LIN {X 0,Y 431.61,Z 997.566,A -85,B 0,C 180,E1 -9443.457,E2 -9443.457} C_VEL
LIN {X 0,Y 431.611,Z 1001.678,A -85,B 0,C 180,E1 -9444.864,E2 -9444.864} C_VEL
LIN {X 0,Y 431.653,Z 1004.723,A -85,B 0,C 180,E1 -9446.268,E2 -9446.268} C_VEL
LIN {X 0,Y 431.594,Z 1006.161,A -85,B 0,C 180,E1 -9447.202,E2 -9447.202} C_VEL
LIN {X 0,Y 431.598,Z 1007.192,A -85,B 0,C 180,E1 -9448.135,E2 -9448.135} C_VEL
LIN {X 0,Y 431.588,Z 1007.819,A -85,B 0,C 180,E1 -9449.069,E2 -9449.069} C_VEL
LIN {X 0,Y 431.588,Z 1008.042,A -85,B 0,C 180,E1 -9450.002,E2 -9450.002} C_VEL
LIN {X 0,Y 431.588,Z 1007.817,A -85,B 0,C 180,E1 -9450.935,E2 -9450.935} C_VEL
LIN {X 0,Y 431.598,Z 1007.188,A -85,B 0,C 180,E1 -9451.868,E2 -9451.868} C_VEL
LIN {X 0,Y 431.594,Z 1006.154,A -85,B 0,C 180,E1 -9452.802,E2 -9452.802} C_VEL
LIN {X 0,Y 431.654,Z 1004.714,A -85,B 0,C 180,E1 -9453.736,E2 -9453.736} C_VEL
LIN {X 0,Y 431.613,Z 1001.67,A -85,B 0,C 180,E1 -9455.14,E2 -9455.14} C_VEL
LIN {X 0,Y 431.606,Z 997.241,A -85,B 0,C 180,E1 -9456.642,E2 -9456.642} C_VEL
LIN {X 0,Y 431.759,Z 991.254,A -85,B 0,C 180,E1 -9458.19,E2 -9458.19} C_VEL
LIN {X 0,Y 432.015,Z 984.395,A -85,B 0,C 180,E1 -9459.6,E2 -9459.6} C_VEL
LIN {X 0,Y 432.389,Z 975.91,A -85,B 0,C 180,E1 -9461.012,E2 -9461.012} C_VEL
LIN {X 0,Y 432.869,Z 967.24,A -85,B 0,C 180,E1 -9462.186,E2 -9462.186} C_VEL
LIN {X 0,Y 433.517,Z 957.475,A -85,B 0,C 180,E1 -9463.269,E2 -9463.269} C_VEL
LIN {X 0,Y 434.054,Z 946.027,A -85,B 0,C 180,E1 -9464.297,E2 -9464.297} C_VEL
LIN {X 0,Y 434.832,Z 934.542,A -85,B 0,C 180,E1 -9465.108,E2 -9465.108} C_VEL
LIN {X 0,Y 435.064,Z 925.091,A -85,B 0,C 180,E1 -9465.64,E2 -9465.64} C_VEL
LIN {X 0,Y 433.844,Z 913.102,A -85,B 0,C 180,E1 -9466.206,E2 -9466.206} C_VEL
LIN {X 0,Y 432.617,Z 900.334,A -85,B 0,C 180,E1 -9466.629,E2 -9466.629} C_VEL
LIN {X 0,Y 432.136,Z 896.114,A -85,B 0,C 180,E1 -9466.747,E2 -9466.747} C_VEL
LIN {X 0,Y 432.528,Z 884.888,A -85,B 0,C 180,E1 -9469.537,E2 -9469.537} C_VEL
LIN {X 0,Y 433.063,Z 870.116,A -85,B 0,C 180,E1 -9473.177,E2 -9473.177} C_VEL
LIN {X 0,Y 433.676,Z 856.799,A -85,B 0,C 180,E1 -9476.467,E2 -9476.467} C_VEL
LIN {X 0,Y 434.24,Z 843.307,A -85,B 0,C 180,E1 -9479.848,E2 -9479.848} C_VEL
LIN {X 0,Y 434.896,Z 831.661,A -85,B 0,C 180,E1 -9482.825,E2 -9482.825} C_VEL
LIN {X 0,Y 435.61,Z 820.099,A -85,B 0,C 180,E1 -9485.875,E2 -9485.875} C_VEL
LIN {X 0,Y 435.573,Z 815.433,A -85,B 0,C 180,E1 -9487.162,E2 -9487.162} C_VEL
LIN {X 0,Y 433.512,Z 804.571,A -85,B 0,C 180,E1 -9490.428,E2 -9490.428} C_VEL
LIN {X 0,Y 432.309,Z 798.638,A -85,B 0,C 180,E1 -9492.373,E2 -9492.373} C_VEL
LIN {X 0,Y 432.29,Z 798.641,A -85,B 0,C 180,E1 -9495.672,E2 -9495.672} C_VEL
LIN {X 0,Y 432.307,Z 798.634,A -85,B 0,C 180,E1 -9498.403,E2 -9498.403} C_VEL
LIN {X 0,Y 432.319,Z 798.635,A -85,B 0,C 180,E1 -9501.848,E2 -9501.848} C_VEL
LIN {X 0,Y 432.299,Z 798.637,A -85,B 0,C 180,E1 -9505.319,E2 -9505.319} C_VEL
LIN {X 0,Y 432.304,Z 798.635,A -85,B 0,C 180,E1 -9508.653,E2 -9508.653} C_VEL
LIN {X 0,Y 432.315,Z 798.634,A -85,B 0,C 180,E1 -9511.872,E2 -9511.872} C_VEL
LIN {X 0,Y 432.339,Z 798.63,A -85,B 0,C 180,E1 -9515.552,E2 -9515.552} C_VEL
LIN {X 0,Y 432.324,Z 798.633,A -85,B 0,C 180,E1 -9519.045,E2 -9519.045} C_VEL
LIN {X 0,Y 432.309,Z 798.637,A -85,B 0,C 180,E1 -9522.008,E2 -9522.008} C_VEL
LIN {X 0,Y 432.404,Z 798.783,A -85,B 0,C 180,E1 -9524.157,E2 -9524.157} C_VEL
LIN {X 0,Y 436.113,Z 810.722,A -85,B 0,C 180,E1 -9525.058,E2 -9525.058} C_VEL
LIN {X 0,Y 436.046,Z 817.668,A -85,B 0,C 180,E1 -9525.561,E2 -9525.561} C_VEL
LIN {X 0,Y 435.466,Z 829.477,A -85,B 0,C 180,E1 -9526.585,E2 -9526.585} C_VEL
LIN {X 0,Y 435.048,Z 837.226,A -85,B 0,C 180,E1 -9527.403,E2 -9527.403} C_VEL
LIN {X 0,Y 434.509,Z 846.358,A -85,B 0,C 180,E1 -9528.572,E2 -9528.572} C_VEL
LIN {X 0,Y 433.963,Z 853.786,A -85,B 0,C 180,E1 -9529.738,E2 -9529.738} C_VEL
LIN {X 0,Y 433.565,Z 859.986,A -85,B 0,C 180,E1 -9530.907,E2 -9530.907} C_VEL
LIN {X 0,Y 433.274,Z 864.988,A -85,B 0,C 180,E1 -9532.038,E2 -9532.038} C_VEL
LIN {X 0,Y 432.89,Z 870.144,A -85,B 0,C 180,E1 -9533.475,E2 -9533.475} C_VEL
LIN {X 0,Y 432.557,Z 872.838,A -85,B 0,C 180,E1 -9534.406,E2 -9534.406} C_VEL
LIN {X 0,Y 432.373,Z 876.618,A -85,B 0,C 180,E1 -9536.272,E2 -9536.272} C_VEL
LIN {X 0,Y 432.358,Z 877.984,A -85,B 0,C 180,E1 -9537.205,E2 -9537.205} C_VEL
LIN {X 0,Y 432.125,Z 879.329,A -85,B 0,C 180,E1 -9539.068,E2 -9539.068} C_VEL
LIN {X 0,Y 432.102,Z 879.413,A -85,B 0,C 180,E1 -9540,E2 -9540} C_VEL
LIN {X 0,Y 432.084,Z 879.058,A -85,B 0,C 180,E1 -9540.932,E2 -9540.932} C_VEL
LIN {X 0,Y 432.049,Z 877.179,A -85,B 0,C 180,E1 -9542.797,E2 -9542.797} C_VEL
LIN {X 0,Y 432.264,Z 873.535,A -85,B 0,C 180,E1 -9544.663,E2 -9544.663} C_VEL
LIN {X 0,Y 432.473,Z 869.651,A -85,B 0,C 180,E1 -9546.064,E2 -9546.064} C_VEL
LIN {X 0,Y 432.683,Z 866.517,A -85,B 0,C 180,E1 -9546.997,E2 -9546.997} C_VEL
LIN {X 0,Y 433.036,Z 859.477,A -85,B 0,C 180,E1 -9548.634,E2 -9548.634} C_VEL
LIN {X 0,Y 433.442,Z 851.992,A -85,B 0,C 180,E1 -9550.038,E2 -9550.038} C_VEL
LIN {X 0,Y 433.77,Z 844.169,A -85,B 0,C 180,E1 -9551.211,E2 -9551.211} C_VEL
LIN {X 0,Y 434.175,Z 836.841,A -85,B 0,C 180,E1 -9552.148,E2 -9552.148} C_VEL
LIN {X 0,Y 434.508,Z 829.377,A -85,B 0,C 180,E1 -9552.969,E2 -9552.969} C_VEL
LIN {X 0,Y 435.018,Z 819.285,A -85,B 0,C 180,E1 -9553.905,E2 -9553.905} C_VEL
LIN {X 0,Y 435.317,Z 810.147,A -85,B 0,C 180,E1 -9554.585,E2 -9554.585} C_VEL
LIN {X 0,Y 433.058,Z 801.364,A -85,B 0,C 180,E1 -9555.231,E2 -9555.231} C_VEL
LIN {X 0,Y 432.36,Z 798.632,A -85,B 0,C 180,E1 -9555.437,E2 -9555.437} C_VEL
LIN {X 0,Y 432.322,Z 798.629,A -85,B 0,C 180,E1 -9558.973,E2 -9558.973} C_VEL
LIN {X 0,Y 432.34,Z 798.627,A -85,B 0,C 180,E1 -9562.091,E2 -9562.091} C_VEL
LIN {X 0,Y 432.317,Z 798.629,A -85,B 0,C 180,E1 -9565.003,E2 -9565.003} C_VEL
LIN {X 0,Y 432.341,Z 798.624,A -85,B 0,C 180,E1 -9568.619,E2 -9568.619} C_VEL
LIN {X 0,Y 432.322,Z 798.629,A -85,B 0,C 180,E1 -9571.346,E2 -9571.346} C_VEL
LIN {X 0,Y 432.337,Z 798.626,A -85,B 0,C 180,E1 -9574.678,E2 -9574.678} C_VEL
LIN {X 0,Y 432.327,Z 798.631,A -85,B 0,C 180,E1 -9578.151,E2 -9578.151} C_VEL
LIN {X 0,Y 432.311,Z 798.634,A -85,B 0,C 180,E1 -9581.8,E2 -9581.8} C_VEL
LIN {X 0,Y 432.34,Z 798.63,A -85,B 0,C 180,E1 -9584.347,E2 -9584.347} C_VEL
LIN {X 0,Y 432.323,Z 798.628,A -85,B 0,C 180,E1 -9587.016,E2 -9587.016} C_VEL
LIN {X 0,Y 432.297,Z 798.636,A -85,B 0,C 180,E1 -9589.827,E2 -9589.827} C_VEL
LIN {X 0,Y 432.311,Z 798.629,A -85,B 0,C 180,E1 -9593.021,E2 -9593.021} C_VEL
LIN {X 0,Y 432.364,Z 798.629,A -85,B 0,C 180,E1 -9595.996,E2 -9595.996} C_VEL
LIN {X 0,Y 432.354,Z 798.623,A -85,B 0,C 180,E1 -9599.489,E2 -9599.489} C_VEL
LIN {X 0,Y 432.392,Z 798.619,A -85,B 0,C 180,E1 -9602.927,E2 -9602.927} C_VEL
LIN {X 0,Y 432.372,Z 798.62,A -85,B 0,C 180,E1 -9606.022,E2 -9606.022} C_VEL
LIN {X 0,Y 432.356,Z 798.63,A -85,B 0,C 180,E1 -9609.045,E2 -9609.045} C_VEL
LIN {X 0,Y 432.379,Z 798.63,A -85,B 0,C 180,E1 -9612.01,E2 -9612.01} C_VEL
LIN {X 0,Y 432.44,Z 798.621,A -85,B 0,C 180,E1 -9614.111,E2 -9614.111} C_VEL
LIN {X 0,Y 435.924,Z 810.401,A -85,B 0,C 180,E1 -9614.93,E2 -9614.93} C_VEL
LIN {X 0,Y 436.372,Z 813.53,A -85,B 0,C 180,E1 -9615.164,E2 -9615.164} C_VEL
LIN {X 0,Y 435.861,Z 824.491,A -85,B 0,C 180,E1 -9616.002,E2 -9616.002} C_VEL
LIN {X 0,Y 435.354,Z 834.277,A -85,B 0,C 180,E1 -9616.937,E2 -9616.937} C_VEL
LIN {X 0,Y 434.776,Z 844.12,A -85,B 0,C 180,E1 -9618.105,E2 -9618.105} C_VEL
LIN {X 0,Y 434.088,Z 853.622,A -85,B 0,C 180,E1 -9619.504,E2 -9619.504} C_VEL
LIN {X 0,Y 433.566,Z 861.188,A -85,B 0,C 180,E1 -9620.905,E2 -9620.905} C_VEL
LIN {X 0,Y 433.226,Z 868.087,A -85,B 0,C 180,E1 -9622.542,E2 -9622.542} C_VEL
LIN {X 0,Y 432.742,Z 872.717,A -85,B 0,C 180,E1 -9623.939,E2 -9623.939} C_VEL
LIN {X 0,Y 432.476,Z 876.365,A -85,B 0,C 180,E1 -9625.403,E2 -9625.403} C_VEL
LIN {X 0,Y 431.7,Z 877.955,A -85,B 0,C 180,E1 -9626.155,E2 -9626.155} C_VEL
LIN {X 0,Y 428.768,Z 880.174,A -85,B 0,C 180,E1 -9627.381,E2 -9627.381} C_VEL
LIN {X 0,Y 426.352,Z 881.483,A -85,B 0,C 180,E1 -9628.38,E2 -9628.38} C_VEL
LIN {X 0,Y 425.255,Z 882.129,A -85,B 0,C 180,E1 -9629.292,E2 -9629.292} C_VEL
LIN {X 0,Y 425.232,Z 882.111,A -85,B 0,C 180,E1 -9629.425,E2 -9629.425} C_VEL
LIN {X 0,Y 425.24,Z 882.07,A -85,B 0,C 180,E1 -9630.945,E2 -9630.945} C_VEL
LIN {X 0,Y 425.338,Z 880.562,A -85,B 0,C 180,E1 -9632.84,E2 -9632.84} C_VEL
LIN {X 0,Y 425.331,Z 879.257,A -85,B 0,C 180,E1 -9633.788,E2 -9633.788} C_VEL
LIN {X 0,Y 425.555,Z 876.454,A -85,B 0,C 180,E1 -9635.21,E2 -9635.21} C_VEL
LIN {X 0,Y 426.011,Z 872.627,A -85,B 0,C 180,E1 -9636.63,E2 -9636.63} C_VEL
LIN {X 0,Y 426.347,Z 867.365,A -85,B 0,C 180,E1 -9638.148,E2 -9638.148} C_VEL
LIN {X 0,Y 426.758,Z 860.36,A -85,B 0,C 180,E1 -9639.716,E2 -9639.716} C_VEL
LIN {X 0,Y 427.409,Z 852.341,A -85,B 0,C 180,E1 -9641.138,E2 -9641.138} C_VEL
LIN {X 0,Y 427.981,Z 844.123,A -85,B 0,C 180,E1 -9642.324,E2 -9642.324} C_VEL
LIN {X 0,Y 428.551,Z 833.96,A -85,B 0,C 180,E1 -9643.513,E2 -9643.513} C_VEL
LIN {X 0,Y 429.309,Z 822.959,A -85,B 0,C 180,E1 -9644.532,E2 -9644.532} C_VEL
LIN {X 0,Y 429.589,Z 814.542,A -85,B 0,C 180,E1 -9645.172,E2 -9645.172} C_VEL
LIN {X 0,Y 427.365,Z 806.003,A -85,B 0,C 180,E1 -9645.825,E2 -9645.825} C_VEL
LIN {X 0,Y 425.38,Z 799.499,A -85,B 0,C 180,E1 -9646.279,E2 -9646.279} C_VEL
LIN {X 0,Y 425.327,Z 799.505,A -85,B 0,C 180,E1 -9649.634,E2 -9649.634} C_VEL
LIN {X 0,Y 425.304,Z 799.506,A -85,B 0,C 180,E1 -9653.363,E2 -9653.363} C_VEL
LIN {X 0,Y 425.344,Z 799.499,A -85,B 0,C 180,E1 -9656.842,E2 -9656.842} C_VEL
LIN {X 0,Y 425.286,Z 799.511,A -85,B 0,C 180,E1 -9659.717,E2 -9659.717} C_VEL
LIN {X 0,Y 425.276,Z 799.508,A -85,B 0,C 180,E1 -9663.046,E2 -9663.046} C_VEL
LIN {X 0,Y 425.277,Z 799.513,A -85,B 0,C 180,E1 -9665.927,E2 -9665.927} C_VEL
LIN {X 0,Y 425.302,Z 799.504,A -85,B 0,C 180,E1 -9669.044,E2 -9669.044} C_VEL
LIN {X 0,Y 425.322,Z 799.505,A -85,B 0,C 180,E1 -9672.644,E2 -9672.644} C_VEL
LIN {X 0,Y 425.324,Z 799.505,A -85,B 0,C 180,E1 -9676.052,E2 -9676.052} C_VEL
LIN {X 0,Y 425.299,Z 799.51,A -85,B 0,C 180,E1 -9678.624,E2 -9678.624} C_VEL
LIN {X 0,Y 425.312,Z 799.5,A -85,B 0,C 180,E1 -9681.103,E2 -9681.103} C_VEL
LIN {X 0,Y 425.287,Z 799.508,A -85,B 0,C 180,E1 -9684.663,E2 -9684.663} C_VEL
LIN {X 0,Y 425.253,Z 799.511,A -85,B 0,C 180,E1 -9688.072,E2 -9688.072} C_VEL
LIN {X 0,Y 425.323,Z 799.502,A -85,B 0,C 180,E1 -9691.367,E2 -9691.367} C_VEL
LIN {X 0,Y 425.281,Z 799.508,A -85,B 0,C 180,E1 -9694.554,E2 -9694.554} C_VEL
LIN {X 0,Y 425.272,Z 799.507,A -85,B 0,C 180,E1 -9697.66,E2 -9697.66} C_VEL
LIN {X 0,Y 425.345,Z 799.5,A -85,B 0,C 180,E1 -9700.703,E2 -9700.703} C_VEL
LIN {X 0,Y 425.371,Z 799.492,A -85,B 0,C 180,E1 -9703.687,E2 -9703.687} C_VEL
LIN {X 0,Y 425.414,Z 799.493,A -85,B 0,C 180,E1 -9707.598,E2 -9707.598} C_VEL
LIN {X 0,Y 425.426,Z 799.492,A -85,B 0,C 180,E1 -9711.45,E2 -9711.45} C_VEL
LIN {X 0,Y 425.533,Z 799.477,A -85,B 0,C 180,E1 -9714.313,E2 -9714.313} C_VEL
LIN {X 0,Y 425.557,Z 799.474,A -85,B 0,C 180,E1 -9718.107,E2 -9718.107} C_VEL
LIN {X 0,Y 425.684,Z 799.46,A -85,B 0,C 180,E1 -9720,E2 -9720} C_VEL
LIN {X 0,Y 425.529,Z 799.478,A -85,B 0,C 180,E1 -9722.84,E2 -9722.84} C_VEL
LIN {X 0,Y 425.522,Z 799.483,A -85,B 0,C 180,E1 -9725.687,E2 -9725.687} C_VEL
LIN {X 0,Y 425.419,Z 799.489,A -85,B 0,C 180,E1 -9728.551,E2 -9728.551} C_VEL
LIN {X 0,Y 425.412,Z 799.488,A -85,B 0,C 180,E1 -9732.402,E2 -9732.402} C_VEL
LIN {X 0,Y 425.37,Z 799.499,A -85,B 0,C 180,E1 -9736.312,E2 -9736.312} C_VEL
LIN {X 0,Y 425.311,Z 799.508,A -85,B 0,C 180,E1 -9739.636,E2 -9739.636} C_VEL
LIN {X 0,Y 425.271,Z 799.512,A -85,B 0,C 180,E1 -9742.34,E2 -9742.34} C_VEL
LIN {X 0,Y 425.302,Z 799.505,A -85,B 0,C 180,E1 -9744.658,E2 -9744.658} C_VEL
LIN {X 0,Y 425.253,Z 799.51,A -85,B 0,C 180,E1 -9747.564,E2 -9747.564} C_VEL
LIN {X 0,Y 425.275,Z 799.51,A -85,B 0,C 180,E1 -9750.762,E2 -9750.762} C_VEL
LIN {X 0,Y 425.276,Z 799.513,A -85,B 0,C 180,E1 -9754.285,E2 -9754.285} C_VEL
LIN {X 0,Y 425.257,Z 799.512,A -85,B 0,C 180,E1 -9757.697,E2 -9757.697} C_VEL
LIN {X 0,Y 425.229,Z 799.519,A -85,B 0,C 180,E1 -9760.516,E2 -9760.516} C_VEL
LIN {X 0,Y 425.234,Z 799.516,A -85,B 0,C 180,E1 -9763.351,E2 -9763.351} C_VEL
LIN {X 0,Y 425.243,Z 799.516,A -85,B 0,C 180,E1 -9766.045,E2 -9766.045} C_VEL
LIN {X 0,Y 425.278,Z 799.594,A -85,B 0,C 180,E1 -9767.351,E2 -9767.351} C_VEL
LIN {X 0,Y 427.317,Z 809.787,A -85,B 0,C 180,E1 -9770.624,E2 -9770.624} C_VEL
LIN {X 0,Y 428.764,Z 818.043,A -85,B 0,C 180,E1 -9773.105,E2 -9773.105} C_VEL
LIN {X 0,Y 428.275,Z 827.154,A -85,B 0,C 180,E1 -9775.596,E2 -9775.596} C_VEL
LIN {X 0,Y 427.577,Z 839.005,A -85,B 0,C 180,E1 -9778.729,E2 -9778.729} C_VEL
LIN {X 0,Y 426.802,Z 853.856,A -85,B 0,C 180,E1 -9782.546,E2 -9782.546} C_VEL
LIN {X 0,Y 426.18,Z 867.174,A -85,B 0,C 180,E1 -9785.914,E2 -9785.914} C_VEL
LIN {X 0,Y 425.616,Z 880.253,A -85,B 0,C 180,E1 -9789.208,E2 -9789.208} C_VEL
LIN {X 0,Y 425.144,Z 893.99,A -85,B 0,C 180,E1 -9792.691,E2 -9792.691} C_VEL
LIN {X 0,Y 425.121,Z 895.102,A -85,B 0,C 180,E1 -9792.976,E2 -9792.976} C_VEL
LIN {X 0,Y 426.617,Z 909.537,A -85,B 0,C 180,E1 -9793.424,E2 -9793.424} C_VEL
LIN {X 0,Y 427.477,Z 920.315,A -85,B 0,C 180,E1 -9793.895,E2 -9793.895} C_VEL
LIN {X 0,Y 428.184,Z 927.555,A -85,B 0,C 180,E1 -9794.289,E2 -9794.289} C_VEL
LIN {X 0,Y 427.593,Z 938.835,A -85,B 0,C 180,E1 -9794.999,E2 -9794.999} C_VEL
LIN {X 0,Y 426.877,Z 949.387,A -85,B 0,C 180,E1 -9795.838,E2 -9795.838} C_VEL
LIN {X 0,Y 426.261,Z 960.089,A -85,B 0,C 180,E1 -9796.899,E2 -9796.899} C_VEL
LIN {X 0,Y 425.63,Z 969.873,A -85,B 0,C 180,E1 -9798.09,E2 -9798.09} C_VEL
LIN {X 0,Y 425.163,Z 977.922,A -85,B 0,C 180,E1 -9799.285,E2 -9799.285} C_VEL
LIN {X 0,Y 424.833,Z 985.824,A -85,B 0,C 180,E1 -9800.72,E2 -9800.72} C_VEL
LIN {X 0,Y 424.627,Z 993.128,A -85,B 0,C 180,E1 -9802.393,E2 -9802.393} C_VEL
LIN {X 0,Y 424.569,Z 997.473,A -85,B 0,C 180,E1 -9803.653,E2 -9803.653} C_VEL
LIN {X 0,Y 424.583,Z 1001.753,A -85,B 0,C 180,E1 -9805.254,E2 -9805.254} C_VEL
LIN {X 0,Y 424.619,Z 1003.688,A -85,B 0,C 180,E1 -9806.206,E2 -9806.206} C_VEL
LIN {X 0,Y 424.558,Z 1005.127,A -85,B 0,C 180,E1 -9807.155,E2 -9807.155} C_VEL
LIN {X 0,Y 424.565,Z 1006.159,A -85,B 0,C 180,E1 -9808.104,E2 -9808.104} C_VEL
LIN {X 0,Y 424.561,Z 1006.788,A -85,B 0,C 180,E1 -9809.053,E2 -9809.053} C_VEL
LIN {X 0,Y 424.564,Z 1007.011,A -85,B 0,C 180,E1 -9810.002,E2 -9810.002} C_VEL
LIN {X 0,Y 424.561,Z 1006.785,A -85,B 0,C 180,E1 -9810.95,E2 -9810.95} C_VEL
LIN {X 0,Y 424.565,Z 1006.155,A -85,B 0,C 180,E1 -9811.899,E2 -9811.899} C_VEL
LIN {X 0,Y 424.559,Z 1005.12,A -85,B 0,C 180,E1 -9812.848,E2 -9812.848} C_VEL
LIN {X 0,Y 424.62,Z 1003.679,A -85,B 0,C 180,E1 -9813.798,E2 -9813.798} C_VEL
LIN {X 0,Y 424.557,Z 1000.629,A -85,B 0,C 180,E1 -9815.225,E2 -9815.225} C_VEL
LIN {X 0,Y 424.543,Z 996.512,A -85,B 0,C 180,E1 -9816.656,E2 -9816.656} C_VEL
LIN {X 0,Y 424.712,Z 990.208,A -85,B 0,C 180,E1 -9818.327,E2 -9818.327} C_VEL
LIN {X 0,Y 424.959,Z 983.343,A -85,B 0,C 180,E1 -9819.761,E2 -9819.761} C_VEL
LIN {X 0,Y 425.374,Z 974.859,A -85,B 0,C 180,E1 -9821.196,E2 -9821.196} C_VEL
LIN {X 0,Y 425.902,Z 966.191,A -85,B 0,C 180,E1 -9822.389,E2 -9822.389} C_VEL
LIN {X 0,Y 426.443,Z 957.878,A -85,B 0,C 180,E1 -9823.341,E2 -9823.341} C_VEL
LIN {X 0,Y 427.03,Z 946.418,A -85,B 0,C 180,E1 -9824.415,E2 -9824.415} C_VEL
LIN {X 0,Y 427.807,Z 935.27,A -85,B 0,C 180,E1 -9825.241,E2 -9825.241} C_VEL
LIN {X 0,Y 428.158,Z 926.328,A -85,B 0,C 180,E1 -9825.777,E2 -9825.777} C_VEL
LIN {X 0,Y 426.957,Z 913.942,A -85,B 0,C 180,E1 -9826.399,E2 -9826.399} C_VEL
LIN {X 0,Y 425.761,Z 900.987,A -85,B 0,C 180,E1 -9826.862,E2 -9826.862} C_VEL
LIN {X 0,Y 425.115,Z 895.012,A -85,B 0,C 180,E1 -9827.05,E2 -9827.05} C_VEL
LIN {X 0,Y 425.554,Z 882.226,A -85,B 0,C 180,E1 -9830.294,E2 -9830.294} C_VEL
LIN {X 0,Y 426.117,Z 868.143,A -85,B 0,C 180,E1 -9833.835,E2 -9833.835} C_VEL
LIN {X 0,Y 426.762,Z 854.761,A -85,B 0,C 180,E1 -9837.216,E2 -9837.216} C_VEL
LIN {X 0,Y 427.385,Z 841.39,A -85,B 0,C 180,E1 -9840.65,E2 -9840.65} C_VEL
LIN {X 0,Y 428.052,Z 830.609,A -85,B 0,C 180,E1 -9843.472,E2 -9843.472} C_VEL
LIN {X 0,Y 428.715,Z 820.618,A -85,B 0,C 180,E1 -9846.169,E2 -9846.169} C_VEL
LIN {X 0,Y 428.554,Z 816.434,A -85,B 0,C 180,E1 -9847.358,E2 -9847.358} C_VEL
LIN {X 0,Y 426.73,Z 806.717,A -85,B 0,C 180,E1 -9850.328,E2 -9850.328} C_VEL
LIN {X 0,Y 425.251,Z 799.518,A -85,B 0,C 180,E1 -9852.728,E2 -9852.728} C_VEL
LIN {X 0,Y 425.254,Z 799.517,A -85,B 0,C 180,E1 -9855.289,E2 -9855.289} C_VEL
LIN {X 0,Y 425.248,Z 799.513,A -85,B 0,C 180,E1 -9858.618,E2 -9858.618} C_VEL
LIN {X 0,Y 425.269,Z 799.511,A -85,B 0,C 180,E1 -9862.305,E2 -9862.305} C_VEL
LIN {X 0,Y 425.272,Z 799.511,A -85,B 0,C 180,E1 -9865.814,E2 -9865.814} C_VEL
LIN {X 0,Y 425.29,Z 799.509,A -85,B 0,C 180,E1 -9869.241,E2 -9869.241} C_VEL
LIN {X 0,Y 425.296,Z 799.508,A -85,B 0,C 180,E1 -9871.365,E2 -9871.365} C_VEL
LIN {X 0,Y 425.242,Z 799.516,A -85,B 0,C 180,E1 -9874.551,E2 -9874.551} C_VEL
LIN {X 0,Y 425.294,Z 799.508,A -85,B 0,C 180,E1 -9877.731,E2 -9877.731} C_VEL
LIN {X 0,Y 425.306,Z 799.511,A -85,B 0,C 180,E1 -9880.701,E2 -9880.701} C_VEL
LIN {X 0,Y 425.334,Z 799.632,A -85,B 0,C 180,E1 -9883.809,E2 -9883.809} C_VEL
LIN {X 0,Y 429.422,Z 812.519,A -85,B 0,C 180,E1 -9884.82,E2 -9884.82} C_VEL
LIN {X 0,Y 429.107,Z 823.295,A -85,B 0,C 180,E1 -9885.657,E2 -9885.657} C_VEL
LIN {X 0,Y 428.656,Z 832.154,A -85,B 0,C 180,E1 -9886.489,E2 -9886.489} C_VEL
LIN {X 0,Y 428.284,Z 838.712,A -85,B 0,C 180,E1 -9887.201,E2 -9887.201} C_VEL
LIN {X 0,Y 427.702,Z 847.782,A -85,B 0,C 180,E1 -9888.387,E2 -9888.387} C_VEL
LIN {X 0,Y 427.126,Z 855.153,A -85,B 0,C 180,E1 -9889.572,E2 -9889.572} C_VEL
LIN {X 0,Y 426.698,Z 861.311,A -85,B 0,C 180,E1 -9890.759,E2 -9890.759} C_VEL
LIN {X 0,Y 426.381,Z 866.058,A -85,B 0,C 180,E1 -9891.849,E2 -9891.849} C_VEL
LIN {X 0,Y 425.95,Z 871.403,A -85,B 0,C 180,E1 -9893.368,E2 -9893.368} C_VEL
LIN {X 0,Y 425.599,Z 874.069,A -85,B 0,C 180,E1 -9894.314,E2 -9894.314} C_VEL
LIN {X 0,Y 425.527,Z 876.127,A -85,B 0,C 180,E1 -9895.263,E2 -9895.263} C_VEL
LIN {X 0,Y 425.372,Z 879.145,A -85,B 0,C 180,E1 -9897.159,E2 -9897.159} C_VEL
LIN {X 0,Y 425.123,Z 880.447,A -85,B 0,C 180,E1 -9899.053,E2 -9899.053} C_VEL
LIN {X 0,Y 425.096,Z 880.505,A -85,B 0,C 180,E1 -9900,E2 -9900} C_VEL
LIN {X 0,Y 425.084,Z 880.121,A -85,B 0,C 180,E1 -9900.947,E2 -9900.947} C_VEL
LIN {X 0,Y 425.031,Z 878.196,A -85,B 0,C 180,E1 -9902.843,E2 -9902.843} C_VEL
LIN {X 0,Y 425.21,Z 875.62,A -85,B 0,C 180,E1 -9904.266,E2 -9904.266} C_VEL
LIN {X 0,Y 425.399,Z 872.051,A -85,B 0,C 180,E1 -9905.689,E2 -9905.689} C_VEL
LIN {X 0,Y 425.692,Z 867.373,A -85,B 0,C 180,E1 -9907.113,E2 -9907.113} C_VEL
LIN {X 0,Y 425.986,Z 861.432,A -85,B 0,C 180,E1 -9908.539,E2 -9908.539} C_VEL
LIN {X 0,Y 426.412,Z 854.062,A -85,B 0,C 180,E1 -9909.966,E2 -9909.966} C_VEL
LIN {X 0,Y 426.756,Z 846.484,A -85,B 0,C 180,E1 -9911.157,E2 -9911.157} C_VEL
LIN {X 0,Y 427.215,Z 838.389,A -85,B 0,C 180,E1 -9912.228,E2 -9912.228} C_VEL
LIN {X 0,Y 427.627,Z 829.831,A -85,B 0,C 180,E1 -9913.181,E2 -9913.181} C_VEL
LIN {X 0,Y 428.15,Z 819.651,A -85,B 0,C 180,E1 -9914.133,E2 -9914.133} C_VEL
LIN {X 0,Y 428.427,Z 812.434,A -85,B 0,C 180,E1 -9914.682,E2 -9914.682} C_VEL
LIN {X 0,Y 427.755,Z 808.595,A -85,B 0,C 180,E1 -9914.973,E2 -9914.973} C_VEL
LIN {X 0,Y 425.319,Z 799.509,A -85,B 0,C 180,E1 -9915.638,E2 -9915.638} C_VEL
LIN {X 0,Y 425.306,Z 799.506,A -85,B 0,C 180,E1 -9919.299,E2 -9919.299} C_VEL
LIN {X 0,Y 425.289,Z 799.503,A -85,B 0,C 180,E1 -9922.339,E2 -9922.339} C_VEL
LIN {X 0,Y 425.254,Z 799.513,A -85,B 0,C 180,E1 -9925.448,E2 -9925.448} C_VEL
LIN {X 0,Y 425.305,Z 799.5,A -85,B 0,C 180,E1 -9928.858,E2 -9928.858} C_VEL
LIN {X 0,Y 425.267,Z 799.507,A -85,B 0,C 180,E1 -9931.927,E2 -9931.927} C_VEL
LIN {X 0,Y 425.299,Z 799.504,A -85,B 0,C 180,E1 -9935.336,E2 -9935.336} C_VEL
LIN {X 0,Y 425.282,Z 799.504,A -85,B 0,C 180,E1 -9938.901,E2 -9938.901} C_VEL
LIN {X 0,Y 425.264,Z 799.507,A -85,B 0,C 180,E1 -9942.655,E2 -9942.655} C_VEL
LIN {X 0,Y 425.291,Z 799.505,A -85,B 0,C 180,E1 -9945.283,E2 -9945.283} C_VEL
LIN {X 0,Y 425.263,Z 799.51,A -85,B 0,C 180,E1 -9948.619,E2 -9948.619} C_VEL
LIN {X 0,Y 425.287,Z 799.506,A -85,B 0,C 180,E1 -9951.099,E2 -9951.099} C_VEL
LIN {X 0,Y 425.304,Z 799.506,A -85,B 0,C 180,E1 -9954.663,E2 -9954.663} C_VEL
LIN {X 0,Y 425.271,Z 799.512,A -85,B 0,C 180,E1 -9958.072,E2 -9958.072} C_VEL
LIN {X 0,Y 425.337,Z 799.495,A -85,B 0,C 180,E1 -9961.367,E2 -9961.367} C_VEL
LIN {X 0,Y 425.29,Z 799.505,A -85,B 0,C 180,E1 -9964.553,E2 -9964.553} C_VEL
LIN {X 0,Y 425.31,Z 799.506,A -85,B 0,C 180,E1 -9966.634,E2 -9966.634} C_VEL
LIN {X 0,Y 425.334,Z 799.509,A -85,B 0,C 180,E1 -9970.363,E2 -9970.363} C_VEL
LIN {X 0,Y 425.419,Z 799.608,A -85,B 0,C 180,E1 -9973.842,E2 -9973.842} C_VEL
LIN {X 0,Y 428.958,Z 811.468,A -85,B 0,C 180,E1 -9974.68,E2 -9974.68} C_VEL
LIN {X 0,Y 429.577,Z 814.669,A -85,B 0,C 180,E1 -9974.931,E2 -9974.931} C_VEL
LIN {X 0,Y 429.056,Z 825.527,A -85,B 0,C 180,E1 -9975.775,E2 -9975.775} C_VEL
LIN {X 0,Y 428.515,Z 835.313,A -85,B 0,C 180,E1 -9976.724,E2 -9976.724} C_VEL
LIN {X 0,Y 427.909,Z 845.154,A -85,B 0,C 180,E1 -9977.911,E2 -9977.911} C_VEL
LIN {X 0,Y 427.184,Z 854.656,A -85,B 0,C 180,E1 -9979.332,E2 -9979.332} C_VEL
LIN {X 0,Y 426.631,Z 862.221,A -85,B 0,C 180,E1 -9980.756,E2 -9980.756} C_VEL
LIN {X 0,Y 426.267,Z 869.119,A -85,B 0,C 180,E1 -9982.419,E2 -9982.419} C_VEL
LIN {X 0,Y 425.762,Z 873.749,A -85,B 0,C 180,E1 -9983.839,E2 -9983.839} C_VEL
LIN {X 0,Y 425.471,Z 877.424,A -85,B 0,C 180,E1 -9985.341,E2 -9985.341} C_VEL
LIN {X 0,Y 425.339,Z 879.091,A -85,B 0,C 180,E1 -9986.209,E2 -9986.209} C_VEL
LIN {X 0,Y 425.341,Z 880.448,A -85,B 0,C 180,E1 -9987.157,E2 -9987.157} C_VEL
LIN {X 0,Y 425.248,Z 882.02,A -85,B 0,C 180,E1 -9989.051,E2 -9989.051} C_VEL
LIN {X 0,Y 425.232,Z 882.111,A -85,B 0,C 180,E1 -9989.425,E2 -9989.425} C_VEL
LIN {X 0,Y 424.57,Z 882.329,A -85,B 0,C 180,E1 -9990.215,E2 -9990.215} C_VEL
LIN {X 0,Y 421.753,Z 882.319,A -85,B 0,C 180,E1 -9991.502,E2 -9991.502} C_VEL
LIN {X 0,Y 419.386,Z 881.821,A -85,B 0,C 180,E1 -9992.536,E2 -9992.536} C_VEL
LIN {X 0,Y 418.384,Z 881.03,A -85,B 0,C 180,E1 -9993.329,E2 -9993.329} C_VEL
LIN {X 0,Y 418.311,Z 880.634,A -85,B 0,C 180,E1 -9993.596,E2 -9993.596} C_VEL
LIN {X 0,Y 418.559,Z 877.484,A -85,B 0,C 180,E1 -9995.297,E2 -9995.297} C_VEL
LIN {X 0,Y 419.041,Z 873.656,A -85,B 0,C 180,E1 -9996.74,E2 -9996.74} C_VEL
LIN {X 0,Y 419.396,Z 868.378,A -85,B 0,C 180,E1 -9998.288,E2 -9998.288} C_VEL
LIN {X 0,Y 419.836,Z 861.389,A -85,B 0,C 180,E1 -9999.878,E2 -9999.878} C_VEL
LIN {X 0,Y 420.528,Z 853.368,A -85,B 0,C 180,E1 -10001.323,E2 -10001.323} C_VEL
LIN {X 0,Y 421.121,Z 845.151,A -85,B 0,C 180,E1 -10002.528,E2 -10002.528} C_VEL
LIN {X 0,Y 421.726,Z 834.987,A -85,B 0,C 180,E1 -10003.736,E2 -10003.736} C_VEL
LIN {X 0,Y 422.51,Z 824.158,A -85,B 0,C 180,E1 -10004.755,E2 -10004.755} C_VEL
LIN {X 0,Y 422.772,Z 815.573,A -85,B 0,C 180,E1 -10005.423,E2 -10005.423} C_VEL
LIN {X 0,Y 419.914,Z 805.598,A -85,B 0,C 180,E1 -10006.2,E2 -10006.2} C_VEL
LIN {X 0,Y 418.34,Z 800.375,A -85,B 0,C 180,E1 -10006.561,E2 -10006.561} C_VEL
LIN {X 0,Y 418.269,Z 800.385,A -85,B 0,C 180,E1 -10009.789,E2 -10009.789} C_VEL
LIN {X 0,Y 418.235,Z 800.384,A -85,B 0,C 180,E1 -10012.734,E2 -10012.734} C_VEL
LIN {X 0,Y 418.267,Z 800.387,A -85,B 0,C 180,E1 -10015.902,E2 -10015.902} C_VEL
LIN {X 0,Y 418.26,Z 800.382,A -85,B 0,C 180,E1 -10019.16,E2 -10019.16} C_VEL
LIN {X 0,Y 418.251,Z 800.383,A -85,B 0,C 180,E1 -10022.842,E2 -10022.842} C_VEL
LIN {X 0,Y 418.241,Z 800.39,A -85,B 0,C 180,E1 -10026.237,E2 -10026.237} C_VEL
LIN {X 0,Y 418.256,Z 800.384,A -85,B 0,C 180,E1 -10029.678,E2 -10029.678} C_VEL
LIN {X 0,Y 418.276,Z 800.386,A -85,B 0,C 180,E1 -10032.328,E2 -10032.328} C_VEL
LIN {X 0,Y 418.264,Z 800.381,A -85,B 0,C 180,E1 -10035.112,E2 -10035.112} C_VEL
LIN {X 0,Y 418.281,Z 800.376,A -85,B 0,C 180,E1 -10037.772,E2 -10037.772} C_VEL
LIN {X 0,Y 418.255,Z 800.378,A -85,B 0,C 180,E1 -10041.558,E2 -10041.558} C_VEL
LIN {X 0,Y 418.247,Z 800.38,A -85,B 0,C 180,E1 -10045.158,E2 -10045.158} C_VEL
LIN {X 0,Y 418.232,Z 800.384,A -85,B 0,C 180,E1 -10047.471,E2 -10047.471} C_VEL
LIN {X 0,Y 418.263,Z 800.386,A -85,B 0,C 180,E1 -10050.892,E2 -10050.892} C_VEL
LIN {X 0,Y 418.256,Z 800.38,A -85,B 0,C 180,E1 -10054.095,E2 -10054.095} C_VEL
LIN {X 0,Y 418.222,Z 800.388,A -85,B 0,C 180,E1 -10057.263,E2 -10057.263} C_VEL
LIN {X 0,Y 418.267,Z 800.379,A -85,B 0,C 180,E1 -10060.363,E2 -10060.363} C_VEL
LIN {X 0,Y 418.3,Z 800.375,A -85,B 0,C 180,E1 -10063.404,E2 -10063.404} C_VEL
LIN {X 0,Y 418.339,Z 800.375,A -85,B 0,C 180,E1 -10066.993,E2 -10066.993} C_VEL
LIN {X 0,Y 418.345,Z 800.367,A -85,B 0,C 180,E1 -10070.329,E2 -10070.329} C_VEL
LIN {X 0,Y 418.472,Z 800.362,A -85,B 0,C 180,E1 -10073.249,E2 -10073.249} C_VEL
LIN {X 0,Y 418.321,Z 800.381,A -85,B 0,C 180,E1 -10075.181,E2 -10075.181} C_VEL
LIN {X 0,Y 418.526,Z 800.35,A -85,B 0,C 180,E1 -10078.075,E2 -10078.075} C_VEL
LIN {X 0,Y 418.654,Z 800.336,A -85,B 0,C 180,E1 -10080,E2 -10080} C_VEL
LIN {X 0,Y 418.484,Z 800.356,A -85,B 0,C 180,E1 -10082.888,E2 -10082.888} C_VEL
LIN {X 0,Y 418.48,Z 800.359,A -85,B 0,C 180,E1 -10085.783,E2 -10085.783} C_VEL
LIN {X 0,Y 418.379,Z 800.366,A -85,B 0,C 180,E1 -10088.696,E2 -10088.696} C_VEL
LIN {X 0,Y 418.314,Z 800.378,A -85,B 0,C 180,E1 -10091.631,E2 -10091.631} C_VEL
LIN {X 0,Y 418.287,Z 800.379,A -85,B 0,C 180,E1 -10094.598,E2 -10094.598} C_VEL
LIN {X 0,Y 418.268,Z 800.385,A -85,B 0,C 180,E1 -10097.605,E2 -10097.605} C_VEL
LIN {X 0,Y 418.233,Z 800.387,A -85,B 0,C 180,E1 -10100.664,E2 -10100.664} C_VEL
LIN {X 0,Y 418.257,Z 800.386,A -85,B 0,C 180,E1 -10103.783,E2 -10103.783} C_VEL
LIN {X 0,Y 418.209,Z 800.386,A -85,B 0,C 180,E1 -10107.049,E2 -10107.049} C_VEL
LIN {X 0,Y 418.227,Z 800.389,A -85,B 0,C 180,E1 -10110.274,E2 -10110.274} C_VEL
LIN {X 0,Y 418.218,Z 800.388,A -85,B 0,C 180,E1 -10113.68,E2 -10113.68} C_VEL
LIN {X 0,Y 418.22,Z 800.388,A -85,B 0,C 180,E1 -10117.226,E2 -10117.226} C_VEL
LIN {X 0,Y 418.194,Z 800.394,A -85,B 0,C 180,E1 -10120.869,E2 -10120.869} C_VEL
LIN {X 0,Y 418.19,Z 800.394,A -85,B 0,C 180,E1 -10123.73,E2 -10123.73} C_VEL
LIN {X 0,Y 418.242,Z 800.532,A -85,B 0,C 180,E1 -10127.016,E2 -10127.016} C_VEL
LIN {X 0,Y 419.969,Z 809.024,A -85,B 0,C 180,E1 -10129.824,E2 -10129.824} C_VEL
LIN {X 0,Y 421.633,Z 817.727,A -85,B 0,C 180,E1 -10132.529,E2 -10132.529} C_VEL
LIN {X 0,Y 421.761,Z 821.912,A -85,B 0,C 180,E1 -10133.735,E2 -10133.735} C_VEL
LIN {X 0,Y 420.91,Z 834.334,A -85,B 0,C 180,E1 -10137.138,E2 -10137.138} C_VEL
LIN {X 0,Y 420.117,Z 846.8,A -85,B 0,C 180,E1 -10140.446,E2 -10140.446} C_VEL
LIN {X 0,Y 419.525,Z 859.083,A -85,B 0,C 180,E1 -10143.647,E2 -10143.647} C_VEL
LIN {X 0,Y 418.891,Z 872.253,A -85,B 0,C 180,E1 -10147.043,E2 -10147.043} C_VEL
LIN {X 0,Y 418.353,Z 885.167,A -85,B 0,C 180,E1 -10150.37,E2 -10150.37} C_VEL
LIN {X 0,Y 418.053,Z 894.045,A -85,B 0,C 180,E1 -10152.677,E2 -10152.677} C_VEL
LIN {X 0,Y 419.651,Z 909.295,A -85,B 0,C 180,E1 -10153.168,E2 -10153.168} C_VEL
LIN {X 0,Y 420.646,Z 921.824,A -85,B 0,C 180,E1 -10153.751,E2 -10153.751} C_VEL
LIN {X 0,Y 421.167,Z 928.544,A -85,B 0,C 180,E1 -10154.144,E2 -10154.144} C_VEL
LIN {X 0,Y 420.446,Z 940.984,A -85,B 0,C 180,E1 -10154.986,E2 -10154.986} C_VEL
LIN {X 0,Y 419.715,Z 952.121,A -85,B 0,C 180,E1 -10155.951,E2 -10155.951} C_VEL
LIN {X 0,Y 419.191,Z 961.373,A -85,B 0,C 180,E1 -10156.941,E2 -10156.941} C_VEL
LIN {X 0,Y 418.542,Z 970.545,A -85,B 0,C 180,E1 -10158.132,E2 -10158.132} C_VEL
LIN {X 0,Y 417.984,Z 979.68,A -85,B 0,C 180,E1 -10159.588,E2 -10159.588} C_VEL
LIN {X 0,Y 417.694,Z 987.075,A -85,B 0,C 180,E1 -10161.048,E2 -10161.048} C_VEL
LIN {X 0,Y 417.563,Z 992.082,A -85,B 0,C 180,E1 -10162.264,E2 -10162.264} C_VEL
LIN {X 0,Y 417.525,Z 996.658,A -85,B 0,C 180,E1 -10163.619,E2 -10163.619} C_VEL
LIN {X 0,Y 417.543,Z 1000.716,A -85,B 0,C 180,E1 -10165.174,E2 -10165.174} C_VEL
LIN {X 0,Y 417.586,Z 1002.654,A -85,B 0,C 180,E1 -10166.142,E2 -10166.142} C_VEL
LIN {X 0,Y 417.522,Z 1004.093,A -85,B 0,C 180,E1 -10167.107,E2 -10167.107} C_VEL
LIN {X 0,Y 417.531,Z 1005.126,A -85,B 0,C 180,E1 -10168.073,E2 -10168.073} C_VEL
LIN {X 0,Y 417.533,Z 1005.756,A -85,B 0,C 180,E1 -10169.037,E2 -10169.037} C_VEL
LIN {X 0,Y 417.539,Z 1005.98,A -85,B 0,C 180,E1 -10170.002,E2 -10170.002} C_VEL
LIN {X 0,Y 417.533,Z 1005.753,A -85,B 0,C 180,E1 -10170.966,E2 -10170.966} C_VEL
LIN {X 0,Y 417.531,Z 1005.121,A -85,B 0,C 180,E1 -10171.931,E2 -10171.931} C_VEL
LIN {X 0,Y 417.523,Z 1004.086,A -85,B 0,C 180,E1 -10172.896,E2 -10172.896} C_VEL
LIN {X 0,Y 417.587,Z 1002.644,A -85,B 0,C 180,E1 -10173.862,E2 -10173.862} C_VEL
LIN {X 0,Y 417.504,Z 999.589,A -85,B 0,C 180,E1 -10175.314,E2 -10175.314} C_VEL
LIN {X 0,Y 417.478,Z 995.467,A -85,B 0,C 180,E1 -10176.769,E2 -10176.769} C_VEL
LIN {X 0,Y 417.644,Z 989.158,A -85,B 0,C 180,E1 -10178.469,E2 -10178.469} C_VEL
LIN {X 0,Y 417.916,Z 982.292,A -85,B 0,C 180,E1 -10179.927,E2 -10179.927} C_VEL
LIN {X 0,Y 418.344,Z 973.805,A -85,B 0,C 180,E1 -10181.386,E2 -10181.386} C_VEL
LIN {X 0,Y 418.95,Z 965.144,A -85,B 0,C 180,E1 -10182.598,E2 -10182.598} C_VEL
LIN {X 0,Y 419.557,Z 954.7,A -85,B 0,C 180,E1 -10183.787,E2 -10183.787} C_VEL
LIN {X 0,Y 420.198,Z 943.919,A -85,B 0,C 180,E1 -10184.779,E2 -10184.779} C_VEL
LIN {X 0,Y 421.014,Z 932.43,A -85,B 0,C 180,E1 -10185.617,E2 -10185.617} C_VEL
LIN {X 0,Y 421.095,Z 926.389,A -85,B 0,C 180,E1 -10185.986,E2 -10185.986} C_VEL
LIN {X 0,Y 420.012,Z 914.055,A -85,B 0,C 180,E1 -10186.63,E2 -10186.63} C_VEL
LIN {X 0,Y 418.844,Z 901.054,A -85,B 0,C 180,E1 -10187.117,E2 -10187.117} C_VEL
LIN {X 0,Y 418.057,Z 894.051,A -85,B 0,C 180,E1 -10187.325,E2 -10187.325} C_VEL
LIN {X 0,Y 418.525,Z 881.23,A -85,B 0,C 180,E1 -10190.65,E2 -10190.65} C_VEL
LIN {X 0,Y 419.122,Z 867.191,A -85,B 0,C 180,E1 -10194.258,E2 -10194.258} C_VEL
LIN {X 0,Y 419.739,Z 854.831,A -85,B 0,C 180,E1 -10197.449,E2 -10197.449} C_VEL
LIN {X 0,Y 420.522,Z 840.512,A -85,B 0,C 180,E1 -10201.206,E2 -10201.206} C_VEL
LIN {X 0,Y 421.327,Z 828.05,A -85,B 0,C 180,E1 -10204.553,E2 -10204.553} C_VEL
LIN {X 0,Y 421.792,Z 819.678,A -85,B 0,C 180,E1 -10206.89,E2 -10206.89} C_VEL
LIN {X 0,Y 420.763,Z 813.3,A -85,B 0,C 180,E1 -10208.82,E2 -10208.82} C_VEL
LIN {X 0,Y 419.031,Z 804.339,A -85,B 0,C 180,E1 -10211.69,E2 -10211.69} C_VEL
LIN {X 0,Y 418.217,Z 800.39,A -85,B 0,C 180,E1 -10213.066,E2 -10213.066} C_VEL
LIN {X 0,Y 418.161,Z 800.398,A -85,B 0,C 180,E1 -10216.279,E2 -10216.279} C_VEL
LIN {X 0,Y 418.21,Z 800.393,A -85,B 0,C 180,E1 -10219.134,E2 -10219.134} C_VEL
LIN {X 0,Y 418.23,Z 800.387,A -85,B 0,C 180,E1 -10222.775,E2 -10222.775} C_VEL
LIN {X 0,Y 418.223,Z 800.39,A -85,B 0,C 180,E1 -10226.32,E2 -10226.32} C_VEL
LIN {X 0,Y 418.238,Z 800.388,A -85,B 0,C 180,E1 -10229.727,E2 -10229.727} C_VEL
LIN {X 0,Y 418.199,Z 800.391,A -85,B 0,C 180,E1 -10233.016,E2 -10233.016} C_VEL
LIN {X 0,Y 418.225,Z 800.391,A -85,B 0,C 180,E1 -10236.215,E2 -10236.215} C_VEL
LIN {X 0,Y 418.228,Z 800.389,A -85,B 0,C 180,E1 -10239.336,E2 -10239.336} C_VEL
LIN {X 0,Y 418.218,Z 800.393,A -85,B 0,C 180,E1 -10242.393,E2 -10242.393} C_VEL
LIN {X 0,Y 418.294,Z 800.417,A -85,B 0,C 180,E1 -10243.435,E2 -10243.435} C_VEL
LIN {X 0,Y 422.381,Z 812.94,A -85,B 0,C 180,E1 -10244.437,E2 -10244.437} C_VEL
LIN {X 0,Y 422.892,Z 815.882,A -85,B 0,C 180,E1 -10244.694,E2 -10244.694} C_VEL
LIN {X 0,Y 422.425,Z 825.003,A -85,B 0,C 180,E1 -10245.422,E2 -10245.422} C_VEL
LIN {X 0,Y 421.915,Z 833.791,A -85,B 0,C 180,E1 -10246.269,E2 -10246.269} C_VEL
LIN {X 0,Y 421.534,Z 840.266,A -85,B 0,C 180,E1 -10246.993,E2 -10246.993} C_VEL
LIN {X 0,Y 420.91,Z 849.268,A -85,B 0,C 180,E1 -10248.197,E2 -10248.197} C_VEL
LIN {X 0,Y 420.305,Z 856.567,A -85,B 0,C 180,E1 -10249.401,E2 -10249.401} C_VEL
LIN {X 0,Y 419.826,Z 862.68,A -85,B 0,C 180,E1 -10250.607,E2 -10250.607} C_VEL
LIN {X 0,Y 419.506,Z 867.112,A -85,B 0,C 180,E1 -10251.64,E2 -10251.64} C_VEL
LIN {X 0,Y 419.015,Z 872.69,A -85,B 0,C 180,E1 -10253.257,E2 -10253.257} C_VEL
LIN {X 0,Y 418.646,Z 875.319,A -85,B 0,C 180,E1 -10254.219,E2 -10254.219} C_VEL
LIN {X 0,Y 418.581,Z 877.359,A -85,B 0,C 180,E1 -10255.184,E2 -10255.184} C_VEL
LIN {X 0,Y 418.383,Z 880.316,A -85,B 0,C 180,E1 -10257.111,E2 -10257.111} C_VEL
LIN {X 0,Y 418.118,Z 881.575,A -85,B 0,C 180,E1 -10259.037,E2 -10259.037} C_VEL
LIN {X 0,Y 418.088,Z 881.601,A -85,B 0,C 180,E1 -10260,E2 -10260} C_VEL
LIN {X 0,Y 418.081,Z 881.184,A -85,B 0,C 180,E1 -10260.963,E2 -10260.963} C_VEL
LIN {X 0,Y 418.012,Z 879.206,A -85,B 0,C 180,E1 -10262.891,E2 -10262.891} C_VEL
LIN {X 0,Y 418.199,Z 876.579,A -85,B 0,C 180,E1 -10264.337,E2 -10264.337} C_VEL
LIN {X 0,Y 418.407,Z 872.951,A -85,B 0,C 180,E1 -10265.784,E2 -10265.784} C_VEL
LIN {X 0,Y 418.702,Z 868.205,A -85,B 0,C 180,E1 -10267.232,E2 -10267.232} C_VEL
LIN {X 0,Y 419.023,Z 862.18,A -85,B 0,C 180,E1 -10268.682,E2 -10268.682} C_VEL
LIN {X 0,Y 419.451,Z 854.75,A -85,B 0,C 180,E1 -10270.133,E2 -10270.133} C_VEL
LIN {X 0,Y 419.811,Z 847.078,A -85,B 0,C 180,E1 -10271.344,E2 -10271.344} C_VEL
LIN {X 0,Y 420.249,Z 839.9,A -85,B 0,C 180,E1 -10272.311,E2 -10272.311} C_VEL
LIN {X 0,Y 420.661,Z 831.434,A -85,B 0,C 180,E1 -10273.281,E2 -10273.281} C_VEL
LIN {X 0,Y 421.17,Z 821.425,A -85,B 0,C 180,E1 -10274.242,E2 -10274.242} C_VEL
LIN {X 0,Y 421.459,Z 812.579,A -85,B 0,C 180,E1 -10274.93,E2 -10274.93} C_VEL
LIN {X 0,Y 419.129,Z 803.703,A -85,B 0,C 180,E1 -10275.613,E2 -10275.613} C_VEL
LIN {X 0,Y 418.297,Z 800.383,A -85,B 0,C 180,E1 -10275.844,E2 -10275.844} C_VEL
LIN {X 0,Y 418.228,Z 800.386,A -85,B 0,C 180,E1 -10279.771,E2 -10279.771} C_VEL
LIN {X 0,Y 418.228,Z 800.382,A -85,B 0,C 180,E1 -10282.737,E2 -10282.737} C_VEL
LIN {X 0,Y 418.214,Z 800.387,A -85,B 0,C 180,E1 -10285.908,E2 -10285.908} C_VEL
LIN {X 0,Y 418.262,Z 800.379,A -85,B 0,C 180,E1 -10289.162,E2 -10289.162} C_VEL
LIN {X 0,Y 418.257,Z 800.374,A -85,B 0,C 180,E1 -10292.842,E2 -10292.842} C_VEL
LIN {X 0,Y 418.245,Z 800.383,A -85,B 0,C 180,E1 -10296.236,E2 -10296.236} C_VEL
LIN {X 0,Y 418.204,Z 800.39,A -85,B 0,C 180,E1 -10299.688,E2 -10299.688} C_VEL
LIN {X 0,Y 418.215,Z 800.388,A -85,B 0,C 180,E1 -10302.317,E2 -10302.317} C_VEL
LIN {X 0,Y 418.242,Z 800.383,A -85,B 0,C 180,E1 -10305.108,E2 -10305.108} C_VEL
LIN {X 0,Y 418.239,Z 800.386,A -85,B 0,C 180,E1 -10307.765,E2 -10307.765} C_VEL
LIN {X 0,Y 418.244,Z 800.385,A -85,B 0,C 180,E1 -10311.556,E2 -10311.556} C_VEL
LIN {X 0,Y 418.264,Z 800.38,A -85,B 0,C 180,E1 -10315.158,E2 -10315.158} C_VEL
LIN {X 0,Y 418.252,Z 800.381,A -85,B 0,C 180,E1 -10317.471,E2 -10317.471} C_VEL
LIN {X 0,Y 418.275,Z 800.376,A -85,B 0,C 180,E1 -10320.895,E2 -10320.895} C_VEL
LIN {X 0,Y 418.268,Z 800.381,A -85,B 0,C 180,E1 -10324.094,E2 -10324.094} C_VEL
LIN {X 0,Y 418.244,Z 800.384,A -85,B 0,C 180,E1 -10327.263,E2 -10327.263} C_VEL
LIN {X 0,Y 418.289,Z 800.387,A -85,B 0,C 180,E1 -10330.363,E2 -10330.363} C_VEL
LIN {X 0,Y 418.335,Z 800.382,A -85,B 0,C 180,E1 -10333.545,E2 -10333.545} C_VEL
LIN {X 0,Y 421.983,Z 812.538,A -85,B 0,C 180,E1 -10334.42,E2 -10334.42} C_VEL
LIN {X 0,Y 422.803,Z 815.809,A -85,B 0,C 180,E1 -10334.691,E2 -10334.691} C_VEL
LIN {X 0,Y 422.25,Z 826.563,A -85,B 0,C 180,E1 -10335.541,E2 -10335.541} C_VEL
LIN {X 0,Y 421.682,Z 836.348,A -85,B 0,C 180,E1 -10336.505,E2 -10336.505} C_VEL
LIN {X 0,Y 421.046,Z 846.188,A -85,B 0,C 180,E1 -10337.711,E2 -10337.711} C_VEL
LIN {X 0,Y 420.284,Z 855.69,A -85,B 0,C 180,E1 -10339.155,E2 -10339.155} C_VEL
LIN {X 0,Y 419.723,Z 863.251,A -85,B 0,C 180,E1 -10340.603,E2 -10340.603} C_VEL
LIN {X 0,Y 419.334,Z 869.134,A -85,B 0,C 180,E1 -10342.01,E2 -10342.01} C_VEL
LIN {X 0,Y 419.035,Z 873.375,A -85,B 0,C 180,E1 -10343.256,E2 -10343.256} C_VEL
LIN {X 0,Y 418.568,Z 877.267,A -85,B 0,C 180,E1 -10344.7,E2 -10344.7} C_VEL
LIN {X 0,Y 418.33,Z 880.123,A -85,B 0,C 180,E1 -10346.145,E2 -10346.145} C_VEL
LIN {X 0,Y 418.327,Z 881.479,A -85,B 0,C 180,E1 -10347.109,E2 -10347.109} C_VEL
LIN {X 0,Y 418.231,Z 883.051,A -85,B 0,C 180,E1 -10349.035,E2 -10349.035} C_VEL
LIN {X 0,Y 418.224,Z 883.28,A -85,B 0,C 180,E1 -10349.998,E2 -10349.998} C_VEL
LIN {X 0,Y 418.234,Z 882.536,A -85,B 0,C 180,E1 -10351.924,E2 -10351.924} C_VEL
LIN {X 0,Y 418.311,Z 880.634,A -85,B 0,C 180,E1 -10353.596,E2 -10353.596} C_VEL
LIN {X 0,Y 417.726,Z 879.496,A -85,B 0,C 180,E1 -10354.386,E2 -10354.386} C_VEL
LIN {X 0,Y 415.175,Z 877.257,A -85,B 0,C 180,E1 -10355.667,E2 -10355.667} C_VEL
LIN {X 0,Y 413.103,Z 874.976,A -85,B 0,C 180,E1 -10356.678,E2 -10356.678} C_VEL
LIN {X 0,Y 412.337,Z 872.847,A -85,B 0,C 180,E1 -10357.436,E2 -10357.436} C_VEL
LIN {X 0,Y 412.342,Z 872.021,A -85,B 0,C 180,E1 -10357.686,E2 -10357.686} C_VEL
LIN {X 0,Y 412.686,Z 865.809,A -85,B 0,C 180,E1 -10359.308,E2 -10359.308} C_VEL
LIN {X 0,Y 413.216,Z 858.631,A -85,B 0,C 180,E1 -10360.781,E2 -10360.781} C_VEL
LIN {X 0,Y 414.039,Z 849.663,A -85,B 0,C 180,E1 -10362.248,E2 -10362.248} C_VEL
LIN {X 0,Y 414.74,Z 839.287,A -85,B 0,C 180,E1 -10363.597,E2 -10363.597} C_VEL
LIN {X 0,Y 415.407,Z 828.691,A -85,B 0,C 180,E1 -10364.699,E2 -10364.699} C_VEL
LIN {X 0,Y 416.008,Z 817.952,A -85,B 0,C 180,E1 -10365.582,E2 -10365.582} C_VEL
LIN {X 0,Y 414.411,Z 811.352,A -85,B 0,C 180,E1 -10366.121,E2 -10366.121} C_VEL
LIN {X 0,Y 411.256,Z 801.258,A -85,B 0,C 180,E1 -10366.887,E2 -10366.887} C_VEL
LIN {X 0,Y 411.228,Z 801.262,A -85,B 0,C 180,E1 -10369.985,E2 -10369.985} C_VEL
LIN {X 0,Y 411.2,Z 801.261,A -85,B 0,C 180,E1 -10373.145,E2 -10373.145} C_VEL
LIN {X 0,Y 411.234,Z 801.259,A -85,B 0,C 180,E1 -10376.379,E2 -10376.379} C_VEL
LIN {X 0,Y 411.195,Z 801.266,A -85,B 0,C 180,E1 -10379.711,E2 -10379.711} C_VEL
LIN {X 0,Y 411.2,Z 801.262,A -85,B 0,C 180,E1 -10383.154,E2 -10383.154} C_VEL
LIN {X 0,Y 411.188,Z 801.266,A -85,B 0,C 180,E1 -10386.551,E2 -10386.551} C_VEL
LIN {X 0,Y 411.219,Z 801.261,A -85,B 0,C 180,E1 -10389.728,E2 -10389.728} C_VEL
LIN {X 0,Y 411.212,Z 801.26,A -85,B 0,C 180,E1 -10393.125,E2 -10393.125} C_VEL
LIN {X 0,Y 411.23,Z 801.259,A -85,B 0,C 180,E1 -10395.869,E2 -10395.869} C_VEL
LIN {X 0,Y 411.202,Z 801.26,A -85,B 0,C 180,E1 -10399.498,E2 -10399.498} C_VEL
LIN {X 0,Y 411.193,Z 801.259,A -85,B 0,C 180,E1 -10402.026,E2 -10402.026} C_VEL
LIN {X 0,Y 411.193,Z 801.257,A -85,B 0,C 180,E1 -10405.665,E2 -10405.665} C_VEL
LIN {X 0,Y 411.184,Z 801.261,A -85,B 0,C 180,E1 -10409.152,E2 -10409.152} C_VEL
LIN {X 0,Y 411.245,Z 801.259,A -85,B 0,C 180,E1 -10412.521,E2 -10412.521} C_VEL
LIN {X 0,Y 411.211,Z 801.258,A -85,B 0,C 180,E1 -10415.783,E2 -10415.783} C_VEL
LIN {X 0,Y 411.18,Z 801.265,A -85,B 0,C 180,E1 -10418.965,E2 -10418.965} C_VEL
LIN {X 0,Y 411.236,Z 801.256,A -85,B 0,C 180,E1 -10422.084,E2 -10422.084} C_VEL
LIN {X 0,Y 411.245,Z 801.255,A -85,B 0,C 180,E1 -10425.147,E2 -10425.147} C_VEL
LIN {X 0,Y 411.285,Z 801.251,A -85,B 0,C 180,E1 -10428.167,E2 -10428.167} C_VEL
LIN {X 0,Y 411.423,Z 801.233,A -85,B 0,C 180,E1 -10432.189,E2 -10432.189} C_VEL
LIN {X 0,Y 411.454,Z 801.232,A -85,B 0,C 180,E1 -10434.118,E2 -10434.118} C_VEL
LIN {X 0,Y 411.495,Z 801.226,A -85,B 0,C 180,E1 -10438.042,E2 -10438.042} C_VEL
LIN {X 0,Y 411.623,Z 801.212,A -85,B 0,C 180,E1 -10440,E2 -10440} C_VEL
LIN {X 0,Y 411.441,Z 801.234,A -85,B 0,C 180,E1 -10442.937,E2 -10442.937} C_VEL
LIN {X 0,Y 411.411,Z 801.234,A -85,B 0,C 180,E1 -10446.868,E2 -10446.868} C_VEL
LIN {X 0,Y 411.29,Z 801.255,A -85,B 0,C 180,E1 -10449.839,E2 -10449.839} C_VEL
LIN {X 0,Y 411.296,Z 801.245,A -85,B 0,C 180,E1 -10453.109,E2 -10453.109} C_VEL
LIN {X 0,Y 411.24,Z 801.257,A -85,B 0,C 180,E1 -10456.889,E2 -10456.889} C_VEL
LIN {X 0,Y 411.214,Z 801.266,A -85,B 0,C 180,E1 -10459.988,E2 -10459.988} C_VEL
LIN {X 0,Y 411.179,Z 801.264,A -85,B 0,C 180,E1 -10463.149,E2 -10463.149} C_VEL
LIN {X 0,Y 411.178,Z 801.266,A -85,B 0,C 180,E1 -10466.385,E2 -10466.385} C_VEL
LIN {X 0,Y 411.182,Z 801.266,A -85,B 0,C 180,E1 -10469.714,E2 -10469.714} C_VEL
LIN {X 0,Y 411.19,Z 801.263,A -85,B 0,C 180,E1 -10473.157,E2 -10473.157} C_VEL
LIN {X 0,Y 411.175,Z 801.268,A -85,B 0,C 180,E1 -10476.553,E2 -10476.553} C_VEL
LIN {X 0,Y 411.154,Z 801.269,A -85,B 0,C 180,E1 -10479.722,E2 -10479.722} C_VEL
LIN {X 0,Y 411.15,Z 801.272,A -85,B 0,C 180,E1 -10483.137,E2 -10483.137} C_VEL
LIN {X 0,Y 411.175,Z 801.415,A -85,B 0,C 180,E1 -10486.656,E2 -10486.656} C_VEL
LIN {X 0,Y 413.033,Z 810.492,A -85,B 0,C 180,E1 -10489.718,E2 -10489.718} C_VEL
LIN {X 0,Y 414.818,Z 820.208,A -85,B 0,C 180,E1 -10492.778,E2 -10492.778} C_VEL
LIN {X 0,Y 414.598,Z 826.045,A -85,B 0,C 180,E1 -10494.456,E2 -10494.456} C_VEL
LIN {X 0,Y 413.67,Z 839.668,A -85,B 0,C 180,E1 -10498.222,E2 -10498.222} C_VEL
LIN {X 0,Y 412.786,Z 853.637,A -85,B 0,C 180,E1 -10501.97,E2 -10501.97} C_VEL
LIN {X 0,Y 412.156,Z 866.277,A -85,B 0,C 180,E1 -10505.308,E2 -10505.308} C_VEL
LIN {X 0,Y 411.487,Z 880.244,A -85,B 0,C 180,E1 -10508.984,E2 -10508.984} C_VEL
LIN {X 0,Y 411.034,Z 892.959,A -85,B 0,C 180,E1 -10512.362,E2 -10512.362} C_VEL
LIN {X 0,Y 412.635,Z 908.368,A -85,B 0,C 180,E1 -10512.878,E2 -10512.878} C_VEL
LIN {X 0,Y 413.525,Z 920.74,A -85,B 0,C 180,E1 -10513.463,E2 -10513.463} C_VEL
LIN {X 0,Y 414.189,Z 929.509,A -85,B 0,C 180,E1 -10513.996,E2 -10513.996} C_VEL
LIN {X 0,Y 413.434,Z 941.498,A -85,B 0,C 180,E1 -10514.851,E2 -10514.851} C_VEL
LIN {X 0,Y 412.682,Z 952.262,A -85,B 0,C 180,E1 -10515.832,E2 -10515.832} C_VEL
LIN {X 0,Y 412.142,Z 960.885,A -85,B 0,C 180,E1 -10516.785,E2 -10516.785} C_VEL
LIN {X 0,Y 411.447,Z 971.163,A -85,B 0,C 180,E1 -10518.174,E2 -10518.174} C_VEL
LIN {X 0,Y 410.894,Z 979.993,A -85,B 0,C 180,E1 -10519.656,E2 -10519.656} C_VEL
LIN {X 0,Y 410.593,Z 987.084,A -85,B 0,C 180,E1 -10521.14,E2 -10521.14} C_VEL
LIN {X 0,Y 410.465,Z 992.791,A -85,B 0,C 180,E1 -10522.624,E2 -10522.624} C_VEL
LIN {X 0,Y 410.42,Z 997.283,A -85,B 0,C 180,E1 -10524.105,E2 -10524.105} C_VEL
LIN {X 0,Y 410.503,Z 999.679,A -85,B 0,C 180,E1 -10525.091,E2 -10525.091} C_VEL
LIN {X 0,Y 410.553,Z 1001.62,A -85,B 0,C 180,E1 -10526.076,E2 -10526.076} C_VEL
LIN {X 0,Y 410.486,Z 1003.059,A -85,B 0,C 180,E1 -10527.058,E2 -10527.058} C_VEL
LIN {X 0,Y 410.497,Z 1004.093,A -85,B 0,C 180,E1 -10528.04,E2 -10528.04} C_VEL
LIN {X 0,Y 410.505,Z 1004.724,A -85,B 0,C 180,E1 -10529.021,E2 -10529.021} C_VEL
LIN {X 0,Y 410.515,Z 1004.948,A -85,B 0,C 180,E1 -10530.002,E2 -10530.002} C_VEL
LIN {X 0,Y 410.505,Z 1004.721,A -85,B 0,C 180,E1 -10530.983,E2 -10530.983} C_VEL
LIN {X 0,Y 410.497,Z 1004.088,A -85,B 0,C 180,E1 -10531.964,E2 -10531.964} C_VEL
LIN {X 0,Y 410.487,Z 1003.051,A -85,B 0,C 180,E1 -10532.946,E2 -10532.946} C_VEL
LIN {X 0,Y 410.555,Z 1001.609,A -85,B 0,C 180,E1 -10533.928,E2 -10533.928} C_VEL
LIN {X 0,Y 410.432,Z 998.545,A -85,B 0,C 180,E1 -10535.406,E2 -10535.406} C_VEL
LIN {X 0,Y 410.427,Z 994.424,A -85,B 0,C 180,E1 -10536.886,E2 -10536.886} C_VEL
LIN {X 0,Y 410.57,Z 988.107,A -85,B 0,C 180,E1 -10538.616,E2 -10538.616} C_VEL
LIN {X 0,Y 410.869,Z 981.24,A -85,B 0,C 180,E1 -10540.099,E2 -10540.099} C_VEL
LIN {X 0,Y 411.339,Z 972.754,A -85,B 0,C 180,E1 -10541.583,E2 -10541.583} C_VEL
LIN {X 0,Y 412.004,Z 964.096,A -85,B 0,C 180,E1 -10542.814,E2 -10542.814} C_VEL
LIN {X 0,Y 412.609,Z 953.403,A -85,B 0,C 180,E1 -10544.049,E2 -10544.049} C_VEL
LIN {X 0,Y 413.343,Z 942.874,A -85,B 0,C 180,E1 -10545.03,E2 -10545.03} C_VEL
LIN {X 0,Y 414.122,Z 931.375,A -85,B 0,C 180,E1 -10545.883,E2 -10545.883} C_VEL
LIN {X 0,Y 414.068,Z 926.361,A -85,B 0,C 180,E1 -10546.202,E2 -10546.202} C_VEL
LIN {X 0,Y 413.066,Z 914.42,A -85,B 0,C 180,E1 -10546.858,E2 -10546.858} C_VEL
LIN {X 0,Y 411.963,Z 901.633,A -85,B 0,C 180,E1 -10547.367,E2 -10547.367} C_VEL
LIN {X 0,Y 411.038,Z 892.97,A -85,B 0,C 180,E1 -10547.64,E2 -10547.64} C_VEL
LIN {X 0,Y 411.475,Z 880.225,A -85,B 0,C 180,E1 -10551.021,E2 -10551.021} C_VEL
LIN {X 0,Y 412.097,Z 867.241,A -85,B 0,C 180,E1 -10554.431,E2 -10554.431} C_VEL
LIN {X 0,Y 412.729,Z 854.887,A -85,B 0,C 180,E1 -10557.691,E2 -10557.691} C_VEL
LIN {X 0,Y 413.508,Z 841.683,A -85,B 0,C 180,E1 -10561.225,E2 -10561.225} C_VEL
LIN {X 0,Y 414.376,Z 829.283,A -85,B 0,C 180,E1 -10564.625,E2 -10564.625} C_VEL
LIN {X 0,Y 414.871,Z 821.649,A -85,B 0,C 180,E1 -10566.784,E2 -10566.784} C_VEL
LIN {X 0,Y 414.312,Z 817.226,A -85,B 0,C 180,E1 -10568.127,E2 -10568.127} C_VEL
LIN {X 0,Y 412.325,Z 807.039,A -85,B 0,C 180,E1 -10571.412,E2 -10571.412} C_VEL
LIN {X 0,Y 411.153,Z 801.267,A -85,B 0,C 180,E1 -10573.421,E2 -10573.421} C_VEL
LIN {X 0,Y 411.109,Z 801.276,A -85,B 0,C 180,E1 -10576.858,E2 -10576.858} C_VEL
LIN {X 0,Y 411.167,Z 801.268,A -85,B 0,C 180,E1 -10580.282,E2 -10580.282} C_VEL
LIN {X 0,Y 411.184,Z 801.265,A -85,B 0,C 180,E1 -10583.451,E2 -10583.451} C_VEL
LIN {X 0,Y 411.208,Z 801.262,A -85,B 0,C 180,E1 -10586.875,E2 -10586.875} C_VEL
LIN {X 0,Y 411.213,Z 801.263,A -85,B 0,C 180,E1 -10590.651,E2 -10590.651} C_VEL
LIN {X 0,Y 411.161,Z 801.269,A -85,B 0,C 180,E1 -10593.614,E2 -10593.614} C_VEL
LIN {X 0,Y 411.178,Z 801.266,A -85,B 0,C 180,E1 -10596.851,E2 -10596.851} C_VEL
LIN {X 0,Y 411.196,Z 801.268,A -85,B 0,C 180,E1 -10600.06,E2 -10600.06} C_VEL
LIN {X 0,Y 411.214,Z 801.264,A -85,B 0,C 180,E1 -10603.032,E2 -10603.032} C_VEL
LIN {X 0,Y 413.488,Z 807.765,A -85,B 0,C 180,E1 -10603.555,E2 -10603.555} C_VEL
LIN {X 0,Y 416.208,Z 816.437,A -85,B 0,C 180,E1 -10604.325,E2 -10604.325} C_VEL
LIN {X 0,Y 415.833,Z 825.386,A -85,B 0,C 180,E1 -10605.047,E2 -10605.047} C_VEL
LIN {X 0,Y 415.278,Z 834.403,A -85,B 0,C 180,E1 -10605.92,E2 -10605.92} C_VEL
LIN {X 0,Y 414.812,Z 841.887,A -85,B 0,C 180,E1 -10606.778,E2 -10606.778} C_VEL
LIN {X 0,Y 414.123,Z 850.817,A -85,B 0,C 180,E1 -10608.001,E2 -10608.001} C_VEL
LIN {X 0,Y 413.486,Z 858.033,A -85,B 0,C 180,E1 -10609.224,E2 -10609.224} C_VEL
LIN {X 0,Y 412.98,Z 864.085,A -85,B 0,C 180,E1 -10610.449,E2 -10610.449} C_VEL
LIN {X 0,Y 412.566,Z 869.097,A -85,B 0,C 180,E1 -10611.675,E2 -10611.675} C_VEL
LIN {X 0,Y 412.088,Z 874.004,A -85,B 0,C 180,E1 -10613.144,E2 -10613.144} C_VEL
LIN {X 0,Y 411.698,Z 876.592,A -85,B 0,C 180,E1 -10614.121,E2 -10614.121} C_VEL
LIN {X 0,Y 411.628,Z 878.613,A -85,B 0,C 180,E1 -10615.103,E2 -10615.103} C_VEL
LIN {X 0,Y 411.392,Z 881.499,A -85,B 0,C 180,E1 -10617.062,E2 -10617.062} C_VEL
LIN {X 0,Y 411.112,Z 882.709,A -85,B 0,C 180,E1 -10619.021,E2 -10619.021} C_VEL
LIN {X 0,Y 411.079,Z 882.697,A -85,B 0,C 180,E1 -10620,E2 -10620} C_VEL
LIN {X 0,Y 411.076,Z 882.25,A -85,B 0,C 180,E1 -10620.98,E2 -10620.98} C_VEL
LIN {X 0,Y 410.993,Z 880.207,A -85,B 0,C 180,E1 -10622.941,E2 -10622.941} C_VEL
LIN {X 0,Y 411.188,Z 877.525,A -85,B 0,C 180,E1 -10624.411,E2 -10624.411} C_VEL
LIN {X 0,Y 411.417,Z 873.831,A -85,B 0,C 180,E1 -10625.883,E2 -10625.883} C_VEL
LIN {X 0,Y 411.713,Z 869.008,A -85,B 0,C 180,E1 -10627.356,E2 -10627.356} C_VEL
LIN {X 0,Y 412.045,Z 862.904,A -85,B 0,C 180,E1 -10628.83,E2 -10628.83} C_VEL
LIN {X 0,Y 412.502,Z 855.406,A -85,B 0,C 180,E1 -10630.305,E2 -10630.305} C_VEL
LIN {X 0,Y 412.866,Z 847.634,A -85,B 0,C 180,E1 -10631.538,E2 -10631.538} C_VEL
LIN {X 0,Y 413.382,Z 839.357,A -85,B 0,C 180,E1 -10632.644,E2 -10632.644} C_VEL
LIN {X 0,Y 413.756,Z 831.79,A -85,B 0,C 180,E1 -10633.507,E2 -10633.507} C_VEL
LIN {X 0,Y 414.29,Z 822.062,A -85,B 0,C 180,E1 -10634.449,E2 -10634.449} C_VEL
LIN {X 0,Y 414.493,Z 813.713,A -85,B 0,C 180,E1 -10635.111,E2 -10635.111} C_VEL
LIN {X 0,Y 411.762,Z 803.325,A -85,B 0,C 180,E1 -10635.91,E2 -10635.91} C_VEL
LIN {X 0,Y 411.249,Z 801.259,A -85,B 0,C 180,E1 -10636.055,E2 -10636.055} C_VEL
LIN {X 0,Y 411.182,Z 801.261,A -85,B 0,C 180,E1 -10639.989,E2 -10639.989} C_VEL
LIN {X 0,Y 411.188,Z 801.26,A -85,B 0,C 180,E1 -10643.149,E2 -10643.149} C_VEL
LIN {X 0,Y 411.169,Z 801.26,A -85,B 0,C 180,E1 -10646.386,E2 -10646.386} C_VEL
LIN {X 0,Y 411.201,Z 801.264,A -85,B 0,C 180,E1 -10649.713,E2 -10649.713} C_VEL
LIN {X 0,Y 411.211,Z 801.252,A -85,B 0,C 180,E1 -10653.156,E2 -10653.156} C_VEL
LIN {X 0,Y 411.194,Z 801.258,A -85,B 0,C 180,E1 -10656.551,E2 -10656.551} C_VEL
LIN {X 0,Y 411.174,Z 801.266,A -85,B 0,C 180,E1 -10659.719,E2 -10659.719} C_VEL
LIN {X 0,Y 411.169,Z 801.262,A -85,B 0,C 180,E1 -10663.134,E2 -10663.134} C_VEL
LIN {X 0,Y 411.174,Z 801.268,A -85,B 0,C 180,E1 -10665.881,E2 -10665.881} C_VEL
LIN {X 0,Y 411.159,Z 801.266,A -85,B 0,C 180,E1 -10668.773,E2 -10668.773} C_VEL
LIN {X 0,Y 411.193,Z 801.268,A -85,B 0,C 180,E1 -10672.025,E2 -10672.025} C_VEL
LIN {X 0,Y 411.211,Z 801.26,A -85,B 0,C 180,E1 -10675.665,E2 -10675.665} C_VEL
LIN {X 0,Y 411.196,Z 801.258,A -85,B 0,C 180,E1 -10679.151,E2 -10679.151} C_VEL
LIN {X 0,Y 411.265,Z 801.252,A -85,B 0,C 180,E1 -10682.521,E2 -10682.521} C_VEL
LIN {X 0,Y 411.223,Z 801.252,A -85,B 0,C 180,E1 -10685.783,E2 -10685.783} C_VEL
LIN {X 0,Y 411.203,Z 801.265,A -85,B 0,C 180,E1 -10688.965,E2 -10688.965} C_VEL
LIN {X 0,Y 411.256,Z 801.263,A -85,B 0,C 180,E1 -10692.084,E2 -10692.084} C_VEL
LIN {X 0,Y 411.309,Z 801.333,A -85,B 0,C 180,E1 -10693.249,E2 -10693.249} C_VEL
LIN {X 0,Y 415.029,Z 813.606,A -85,B 0,C 180,E1 -10694.152,E2 -10694.152} C_VEL
LIN {X 0,Y 416.028,Z 817.633,A -85,B 0,C 180,E1 -10694.493,E2 -10694.493} C_VEL
LIN {X 0,Y 415.391,Z 828.944,A -85,B 0,C 180,E1 -10695.422,E2 -10695.422} C_VEL
LIN {X 0,Y 414.714,Z 839.496,A -85,B 0,C 180,E1 -10696.524,E2 -10696.524} C_VEL
LIN {X 0,Y 414.049,Z 848.967,A -85,B 0,C 180,E1 -10697.749,E2 -10697.749} C_VEL
LIN {X 0,Y 413.388,Z 856.724,A -85,B 0,C 180,E1 -10698.972,E2 -10698.972} C_VEL
LIN {X 0,Y 412.802,Z 864.283,A -85,B 0,C 180,E1 -10700.444,E2 -10700.444} C_VEL
LIN {X 0,Y 412.385,Z 870.154,A -85,B 0,C 180,E1 -10701.871,E2 -10701.871} C_VEL
LIN {X 0,Y 412.064,Z 874.407,A -85,B 0,C 180,E1 -10703.141,E2 -10703.141} C_VEL
LIN {X 0,Y 411.573,Z 878.299,A -85,B 0,C 180,E1 -10704.609,E2 -10704.609} C_VEL
LIN {X 0,Y 411.322,Z 881.155,A -85,B 0,C 180,E1 -10706.079,E2 -10706.079} C_VEL
LIN {X 0,Y 411.312,Z 882.511,A -85,B 0,C 180,E1 -10707.06,E2 -10707.06} C_VEL
LIN {X 0,Y 411.214,Z 884.081,A -85,B 0,C 180,E1 -10709.019,E2 -10709.019} C_VEL
LIN {X 0,Y 411.203,Z 884.311,A -85,B 0,C 180,E1 -10709.998,E2 -10709.998} C_VEL
LIN {X 0,Y 411.233,Z 883.564,A -85,B 0,C 180,E1 -10711.957,E2 -10711.957} C_VEL
LIN {X 0,Y 411.3,Z 881.705,A -85,B 0,C 180,E1 -10713.627,E2 -10713.627} C_VEL
LIN {X 0,Y 411.564,Z 878.515,A -85,B 0,C 180,E1 -10715.387,E2 -10715.387} C_VEL
LIN {X 0,Y 412.071,Z 874.686,A -85,B 0,C 180,E1 -10716.855,E2 -10716.855} C_VEL
LIN {X 0,Y 412.342,Z 872.021,A -85,B 0,C 180,E1 -10717.686,E2 -10717.686} C_VEL
LIN {X 0,Y 411.898,Z 869.544,A -85,B 0,C 180,E1 -10718.43,E2 -10718.43} C_VEL
LIN {X 0,Y 409.35,Z 865.308,A -85,B 0,C 180,E1 -10719.633,E2 -10719.633} C_VEL
LIN {X 0,Y 406.919,Z 860.41,A -85,B 0,C 180,E1 -10720.793,E2 -10720.793} C_VEL
LIN {X 0,Y 406.648,Z 856.898,A -85,B 0,C 180,E1 -10721.458,E2 -10721.458} C_VEL
LIN {X 0,Y 407.318,Z 848.947,A -85,B 0,C 180,E1 -10722.707,E2 -10722.707} C_VEL
LIN {X 0,Y 407.978,Z 839.268,A -85,B 0,C 180,E1 -10723.954,E2 -10723.954} C_VEL
LIN {X 0,Y 408.616,Z 829.717,A -85,B 0,C 180,E1 -10724.949,E2 -10724.949} C_VEL
LIN {X 0,Y 409.231,Z 819.72,A -85,B 0,C 180,E1 -10725.791,E2 -10725.791} C_VEL
LIN {X 0,Y 407.904,Z 813.905,A -85,B 0,C 180,E1 -10726.282,E2 -10726.282} C_VEL
LIN {X 0,Y 404.202,Z 802.138,A -85,B 0,C 180,E1 -10727.19,E2 -10727.19} C_VEL
LIN {X 0,Y 404.162,Z 802.139,A -85,B 0,C 180,E1 -10730.349,E2 -10730.349} C_VEL
LIN {X 0,Y 404.166,Z 802.141,A -85,B 0,C 180,E1 -10733.572,E2 -10733.572} C_VEL
LIN {X 0,Y 404.18,Z 802.141,A -85,B 0,C 180,E1 -10735.764,E2 -10735.764} C_VEL
LIN {X 0,Y 404.191,Z 802.14,A -85,B 0,C 180,E1 -10737.998,E2 -10737.998} C_VEL
LIN {X 0,Y 404.134,Z 802.144,A -85,B 0,C 180,E1 -10741.556,E2 -10741.556} C_VEL
LIN {X 0,Y 404.178,Z 802.136,A -85,B 0,C 180,E1 -10745.014,E2 -10745.014} C_VEL
LIN {X 0,Y 404.155,Z 802.14,A -85,B 0,C 180,E1 -10748.754,E2 -10748.754} C_VEL
LIN {X 0,Y 404.182,Z 802.136,A -85,B 0,C 180,E1 -10751.609,E2 -10751.609} C_VEL
LIN {X 0,Y 404.187,Z 802.14,A -85,B 0,C 180,E1 -10754.528,E2 -10754.528} C_VEL
LIN {X 0,Y 404.2,Z 802.129,A -85,B 0,C 180,E1 -10757.304,E2 -10757.304} C_VEL
LIN {X 0,Y 404.157,Z 802.14,A -85,B 0,C 180,E1 -10759.954,E2 -10759.954} C_VEL
LIN {X 0,Y 404.129,Z 802.143,A -85,B 0,C 180,E1 -10763.122,E2 -10763.122} C_VEL
LIN {X 0,Y 404.132,Z 802.139,A -85,B 0,C 180,E1 -10766.186,E2 -10766.186} C_VEL
LIN {X 0,Y 404.139,Z 802.136,A -85,B 0,C 180,E1 -10769.714,E2 -10769.714} C_VEL
LIN {X 0,Y 404.181,Z 802.136,A -85,B 0,C 180,E1 -10773.122,E2 -10773.122} C_VEL
LIN {X 0,Y 404.162,Z 802.138,A -85,B 0,C 180,E1 -10775.333,E2 -10775.333} C_VEL
LIN {X 0,Y 404.123,Z 802.144,A -85,B 0,C 180,E1 -10778.58,E2 -10778.58} C_VEL
LIN {X 0,Y 404.194,Z 802.134,A -85,B 0,C 180,E1 -10781.761,E2 -10781.761} C_VEL
LIN {X 0,Y 404.191,Z 802.132,A -85,B 0,C 180,E1 -10784.881,E2 -10784.881} C_VEL
LIN {X 0,Y 404.255,Z 802.127,A -85,B 0,C 180,E1 -10787.958,E2 -10787.958} C_VEL
LIN {X 0,Y 404.366,Z 802.113,A -85,B 0,C 180,E1 -10792.007,E2 -10792.007} C_VEL
LIN {X 0,Y 404.403,Z 802.111,A -85,B 0,C 180,E1 -10794.015,E2 -10794.015} C_VEL
LIN {X 0,Y 404.465,Z 802.102,A -85,B 0,C 180,E1 -10798.008,E2 -10798.008} C_VEL
LIN {X 0,Y 404.593,Z 802.088,A -85,B 0,C 180,E1 -10800,E2 -10800} C_VEL
LIN {X 0,Y 404.399,Z 802.112,A -85,B 0,C 180,E1 -10802.989,E2 -10802.989} C_VEL
LIN {X 0,Y 404.361,Z 802.113,A -85,B 0,C 180,E1 -10806.988,E2 -10806.988} C_VEL
LIN {X 0,Y 404.253,Z 802.13,A -85,B 0,C 180,E1 -10810.012,E2 -10810.012} C_VEL
LIN {X 0,Y 404.249,Z 802.124,A -85,B 0,C 180,E1 -10813.212,E2 -10813.212} C_VEL
LIN {X 0,Y 404.199,Z 802.134,A -85,B 0,C 180,E1 -10817.008,E2 -10817.008} C_VEL
LIN {X 0,Y 404.147,Z 802.144,A -85,B 0,C 180,E1 -10820.352,E2 -10820.352} C_VEL
LIN {X 0,Y 404.141,Z 802.143,A -85,B 0,C 180,E1 -10823.576,E2 -10823.576} C_VEL
LIN {X 0,Y 404.118,Z 802.142,A -85,B 0,C 180,E1 -10826.883,E2 -10826.883} C_VEL
LIN {X 0,Y 404.129,Z 802.145,A -85,B 0,C 180,E1 -10830.287,E2 -10830.287} C_VEL
LIN {X 0,Y 404.123,Z 802.145,A -85,B 0,C 180,E1 -10833.814,E2 -10833.814} C_VEL
LIN {X 0,Y 404.118,Z 802.147,A -85,B 0,C 180,E1 -10836.875,E2 -10836.875} C_VEL
LIN {X 0,Y 404.104,Z 802.149,A -85,B 0,C 180,E1 -10840.076,E2 -10840.076} C_VEL
LIN {X 0,Y 404.13,Z 802.147,A -85,B 0,C 180,E1 -10843.084,E2 -10843.084} C_VEL
LIN {X 0,Y 404.14,Z 802.293,A -85,B 0,C 180,E1 -10846.291,E2 -10846.291} C_VEL
LIN {X 0,Y 405.842,Z 810.533,A -85,B 0,C 180,E1 -10849.137,E2 -10849.137} C_VEL
LIN {X 0,Y 407.782,Z 820.756,A -85,B 0,C 180,E1 -10852.448,E2 -10852.448} C_VEL
LIN {X 0,Y 407.903,Z 824.37,A -85,B 0,C 180,E1 -10853.532,E2 -10853.532} C_VEL
LIN {X 0,Y 406.887,Z 837.752,A -85,B 0,C 180,E1 -10857.335,E2 -10857.335} C_VEL
LIN {X 0,Y 405.903,Z 852.116,A -85,B 0,C 180,E1 -10861.286,E2 -10861.286} C_VEL
LIN {X 0,Y 405.261,Z 863.604,A -85,B 0,C 180,E1 -10864.393,E2 -10864.393} C_VEL
LIN {X 0,Y 404.594,Z 875.273,A -85,B 0,C 180,E1 -10867.535,E2 -10867.535} C_VEL
LIN {X 0,Y 404.145,Z 887.03,A -85,B 0,C 180,E1 -10870.709,E2 -10870.709} C_VEL
LIN {X 0,Y 403.972,Z 891.974,A -85,B 0,C 180,E1 -10872.059,E2 -10872.059} C_VEL
LIN {X 0,Y 405.596,Z 906.622,A -85,B 0,C 180,E1 -10872.548,E2 -10872.548} C_VEL
LIN {X 0,Y 406.453,Z 919.662,A -85,B 0,C 180,E1 -10873.167,E2 -10873.167} C_VEL
LIN {X 0,Y 407.272,Z 928.457,A -85,B 0,C 180,E1 -10873.717,E2 -10873.717} C_VEL
LIN {X 0,Y 406.577,Z 940.458,A -85,B 0,C 180,E1 -10874.589,E2 -10874.589} C_VEL
LIN {X 0,Y 405.758,Z 951.216,A -85,B 0,C 180,E1 -10875.585,E2 -10875.585} C_VEL
LIN {X 0,Y 405.104,Z 960.4,A -85,B 0,C 180,E1 -10876.624,E2 -10876.624} C_VEL
LIN {X 0,Y 404.392,Z 970.107,A -85,B 0,C 180,E1 -10877.965,E2 -10877.965} C_VEL
LIN {X 0,Y 403.832,Z 978.94,A -85,B 0,C 180,E1 -10879.473,E2 -10879.473} C_VEL
LIN {X 0,Y 403.538,Z 986.037,A -85,B 0,C 180,E1 -10880.984,E2 -10880.984} C_VEL
LIN {X 0,Y 403.397,Z 991.745,A -85,B 0,C 180,E1 -10882.494,E2 -10882.494} C_VEL
LIN {X 0,Y 403.372,Z 996.243,A -85,B 0,C 180,E1 -10884.001,E2 -10884.001} C_VEL
LIN {X 0,Y 403.437,Z 998.639,A -85,B 0,C 180,E1 -10885.005,E2 -10885.005} C_VEL
LIN {X 0,Y 403.521,Z 1000.585,A -85,B 0,C 180,E1 -10886.007,E2 -10886.007} C_VEL
LIN {X 0,Y 403.45,Z 1002.025,A -85,B 0,C 180,E1 -10887.006,E2 -10887.006} C_VEL
LIN {X 0,Y 403.463,Z 1003.06,A -85,B 0,C 180,E1 -10888.005,E2 -10888.005} C_VEL
LIN {X 0,Y 403.477,Z 1003.692,A -85,B 0,C 180,E1 -10889.004,E2 -10889.004} C_VEL
LIN {X 0,Y 403.49,Z 1003.917,A -85,B 0,C 180,E1 -10890.002,E2 -10890.002} C_VEL
LIN {X 0,Y 403.477,Z 1003.689,A -85,B 0,C 180,E1 -10891,E2 -10891} C_VEL
LIN {X 0,Y 403.463,Z 1003.054,A -85,B 0,C 180,E1 -10891.998,E2 -10891.998} C_VEL
LIN {X 0,Y 403.451,Z 1002.016,A -85,B 0,C 180,E1 -10892.997,E2 -10892.997} C_VEL
LIN {X 0,Y 403.522,Z 1000.573,A -85,B 0,C 180,E1 -10893.997,E2 -10893.997} C_VEL
LIN {X 0,Y 403.365,Z 997.503,A -85,B 0,C 180,E1 -10895.501,E2 -10895.501} C_VEL
LIN {X 0,Y 403.387,Z 993.382,A -85,B 0,C 180,E1 -10897.007,E2 -10897.007} C_VEL
LIN {X 0,Y 403.513,Z 987.057,A -85,B 0,C 180,E1 -10898.768,E2 -10898.768} C_VEL
LIN {X 0,Y 403.802,Z 980.185,A -85,B 0,C 180,E1 -10900.278,E2 -10900.278} C_VEL
LIN {X 0,Y 404.34,Z 971.703,A -85,B 0,C 180,E1 -10901.786,E2 -10901.786} C_VEL
LIN {X 0,Y 405.048,Z 963.046,A -85,B 0,C 180,E1 -10903.038,E2 -10903.038} C_VEL
LIN {X 0,Y 405.656,Z 952.347,A -85,B 0,C 180,E1 -10904.295,E2 -10904.295} C_VEL
LIN {X 0,Y 406.434,Z 941.82,A -85,B 0,C 180,E1 -10905.291,E2 -10905.291} C_VEL
LIN {X 0,Y 407.221,Z 930.316,A -85,B 0,C 180,E1 -10906.16,E2 -10906.16} C_VEL
LIN {X 0,Y 406.394,Z 918.291,A -85,B 0,C 180,E1 -10906.904,E2 -10906.904} C_VEL
LIN {X 0,Y 405.372,Z 904.495,A -85,B 0,C 180,E1 -10907.533,E2 -10907.533} C_VEL
LIN {X 0,Y 403.978,Z 891.902,A -85,B 0,C 180,E1 -10907.962,E2 -10907.962} C_VEL
LIN {X 0,Y 404.434,Z 879.215,A -85,B 0,C 180,E1 -10911.405,E2 -10911.405} C_VEL
LIN {X 0,Y 405.052,Z 867.279,A -85,B 0,C 180,E1 -10914.61,E2 -10914.61} C_VEL
LIN {X 0,Y 405.731,Z 854.93,A -85,B 0,C 180,E1 -10917.943,E2 -10917.943} C_VEL
LIN {X 0,Y 406.618,Z 841.205,A -85,B 0,C 180,E1 -10921.698,E2 -10921.698} C_VEL
LIN {X 0,Y 407.58,Z 828.43,A -85,B 0,C 180,E1 -10925.287,E2 -10925.287} C_VEL
LIN {X 0,Y 407.885,Z 822.238,A -85,B 0,C 180,E1 -10927.091,E2 -10927.091} C_VEL
LIN {X 0,Y 406.731,Z 815.193,A -85,B 0,C 180,E1 -10929.316,E2 -10929.316} C_VEL
LIN {X 0,Y 404.784,Z 805.355,A -85,B 0,C 180,E1 -10932.621,E2 -10932.621} C_VEL
LIN {X 0,Y 404.095,Z 802.146,A -85,B 0,C 180,E1 -10933.756,E2 -10933.756} C_VEL
LIN {X 0,Y 404.071,Z 802.153,A -85,B 0,C 180,E1 -10936.93,E2 -10936.93} C_VEL
LIN {X 0,Y 404.138,Z 802.146,A -85,B 0,C 180,E1 -10939.952,E2 -10939.952} C_VEL
LIN {X 0,Y 404.128,Z 802.145,A -85,B 0,C 180,E1 -10943.128,E2 -10943.128} C_VEL
LIN {X 0,Y 404.169,Z 802.14,A -85,B 0,C 180,E1 -10946.582,E2 -10946.582} C_VEL
LIN {X 0,Y 404.156,Z 802.144,A -85,B 0,C 180,E1 -10950.399,E2 -10950.399} C_VEL
LIN {X 0,Y 404.129,Z 802.146,A -85,B 0,C 180,E1 -10954.23,E2 -10954.23} C_VEL
LIN {X 0,Y 404.167,Z 802.139,A -85,B 0,C 180,E1 -10957.508,E2 -10957.508} C_VEL
LIN {X 0,Y 404.126,Z 802.149,A -85,B 0,C 180,E1 -10960.706,E2 -10960.706} C_VEL
LIN {X 0,Y 404.138,Z 802.146,A -85,B 0,C 180,E1 -10962.602,E2 -10962.602} C_VEL
LIN {X 0,Y 407.874,Z 812.638,A -85,B 0,C 180,E1 -10963.506,E2 -10963.506} C_VEL
LIN {X 0,Y 409.655,Z 818.57,A -85,B 0,C 180,E1 -10964.068,E2 -10964.068} C_VEL
LIN {X 0,Y 409.2,Z 827.186,A -85,B 0,C 180,E1 -10964.784,E2 -10964.784} C_VEL
LIN {X 0,Y 408.581,Z 836.217,A -85,B 0,C 180,E1 -10965.684,E2 -10965.684} C_VEL
LIN {X 0,Y 408.103,Z 843.579,A -85,B 0,C 180,E1 -10966.557,E2 -10966.557} C_VEL
LIN {X 0,Y 407.358,Z 852.426,A -85,B 0,C 180,E1 -10967.799,E2 -10967.799} C_VEL
LIN {X 0,Y 406.68,Z 859.552,A -85,B 0,C 180,E1 -10969.042,E2 -10969.042} C_VEL
LIN {X 0,Y 406.253,Z 864.459,A -85,B 0,C 180,E1 -10970.038,E2 -10970.038} C_VEL
LIN {X 0,Y 405.906,Z 868.715,A -85,B 0,C 180,E1 -10971.035,E2 -10971.035} C_VEL
LIN {X 0,Y 405.169,Z 875.35,A -85,B 0,C 180,E1 -10973.026,E2 -10973.026} C_VEL
LIN {X 0,Y 404.755,Z 877.884,A -85,B 0,C 180,E1 -10974.02,E2 -10974.02} C_VEL
LIN {X 0,Y 404.672,Z 879.89,A -85,B 0,C 180,E1 -10975.018,E2 -10975.018} C_VEL
LIN {X 0,Y 404.402,Z 882.691,A -85,B 0,C 180,E1 -10977.011,E2 -10977.011} C_VEL
LIN {X 0,Y 404.107,Z 883.852,A -85,B 0,C 180,E1 -10979.004,E2 -10979.004} C_VEL
LIN {X 0,Y 404.068,Z 883.794,A -85,B 0,C 180,E1 -10980,E2 -10980} C_VEL
LIN {X 0,Y 404.069,Z 883.314,A -85,B 0,C 180,E1 -10980.997,E2 -10980.997} C_VEL
LIN {X 0,Y 403.972,Z 881.198,A -85,B 0,C 180,E1 -10982.992,E2 -10982.992} C_VEL
LIN {X 0,Y 404.178,Z 878.454,A -85,B 0,C 180,E1 -10984.488,E2 -10984.488} C_VEL
LIN {X 0,Y 404.427,Z 874.689,A -85,B 0,C 180,E1 -10985.985,E2 -10985.985} C_VEL
LIN {X 0,Y 404.724,Z 869.786,A -85,B 0,C 180,E1 -10987.483,E2 -10987.483} C_VEL
LIN {X 0,Y 405.058,Z 863.604,A -85,B 0,C 180,E1 -10988.984,E2 -10988.984} C_VEL
LIN {X 0,Y 405.559,Z 856.031,A -85,B 0,C 180,E1 -10990.484,E2 -10990.484} C_VEL
LIN {X 0,Y 405.929,Z 848.153,A -85,B 0,C 180,E1 -10991.738,E2 -10991.738} C_VEL
LIN {X 0,Y 406.403,Z 840.782,A -85,B 0,C 180,E1 -10992.738,E2 -10992.738} C_VEL
LIN {X 0,Y 406.814,Z 833.288,A -85,B 0,C 180,E1 -10993.614,E2 -10993.614} C_VEL
LIN {X 0,Y 407.374,Z 823.036,A -85,B 0,C 180,E1 -10994.628,E2 -10994.628} C_VEL
LIN {X 0,Y 407.664,Z 815.798,A -85,B 0,C 180,E1 -10995.217,E2 -10995.217} C_VEL
LIN {X 0,Y 405.019,Z 805.327,A -85,B 0,C 180,E1 -10996.048,E2 -10996.048} C_VEL
LIN {X 0,Y 404.201,Z 802.136,A -85,B 0,C 180,E1 -10996.285,E2 -10996.285} C_VEL
LIN {X 0,Y 404.143,Z 802.135,A -85,B 0,C 180,E1 -11000.353,E2 -11000.353} C_VEL
LIN {X 0,Y 404.149,Z 802.142,A -85,B 0,C 180,E1 -11003.576,E2 -11003.576} C_VEL
LIN {X 0,Y 404.136,Z 802.142,A -85,B 0,C 180,E1 -11005.77,E2 -11005.77} C_VEL
LIN {X 0,Y 404.159,Z 802.139,A -85,B 0,C 180,E1 -11009.602,E2 -11009.602} C_VEL
LIN {X 0,Y 404.146,Z 802.132,A -85,B 0,C 180,E1 -11012.621,E2 -11012.621} C_VEL
LIN {X 0,Y 404.152,Z 802.137,A -85,B 0,C 180,E1 -11015.182,E2 -11015.182} C_VEL
LIN {X 0,Y 404.138,Z 802.138,A -85,B 0,C 180,E1 -11018.759,E2 -11018.759} C_VEL
LIN {X 0,Y 404.113,Z 802.145,A -85,B 0,C 180,E1 -11021.596,E2 -11021.596} C_VEL
LIN {X 0,Y 404.15,Z 802.14,A -85,B 0,C 180,E1 -11024.521,E2 -11024.521} C_VEL
LIN {X 0,Y 404.138,Z 802.14,A -85,B 0,C 180,E1 -11027.294,E2 -11027.294} C_VEL
LIN {X 0,Y 404.139,Z 802.143,A -85,B 0,C 180,E1 -11029.95,E2 -11029.95} C_VEL
LIN {X 0,Y 404.141,Z 802.137,A -85,B 0,C 180,E1 -11033.125,E2 -11033.125} C_VEL
LIN {X 0,Y 404.151,Z 802.144,A -85,B 0,C 180,E1 -11036.187,E2 -11036.187} C_VEL
LIN {X 0,Y 404.152,Z 802.137,A -85,B 0,C 180,E1 -11039.714,E2 -11039.714} C_VEL
LIN {X 0,Y 404.2,Z 802.129,A -85,B 0,C 180,E1 -11043.122,E2 -11043.122} C_VEL
LIN {X 0,Y 404.179,Z 802.128,A -85,B 0,C 180,E1 -11045.333,E2 -11045.333} C_VEL
LIN {X 0,Y 404.166,Z 802.144,A -85,B 0,C 180,E1 -11048.581,E2 -11048.581} C_VEL
LIN {X 0,Y 404.214,Z 802.138,A -85,B 0,C 180,E1 -11051.761,E2 -11051.761} C_VEL
LIN {X 0,Y 404.22,Z 802.138,A -85,B 0,C 180,E1 -11052.925,E2 -11052.925} C_VEL
LIN {X 0,Y 408.065,Z 814.677,A -85,B 0,C 180,E1 -11053.874,E2 -11053.874} C_VEL
LIN {X 0,Y 409.064,Z 818.137,A -85,B 0,C 180,E1 -11054.18,E2 -11054.18} C_VEL
LIN {X 0,Y 409.025,Z 824.613,A -85,B 0,C 180,E1 -11054.7,E2 -11054.7} C_VEL
LIN {X 0,Y 408.264,Z 834.968,A -85,B 0,C 180,E1 -11055.671,E2 -11055.671} C_VEL
LIN {X 0,Y 407.586,Z 844.561,A -85,B 0,C 180,E1 -11056.791,E2 -11056.791} C_VEL
LIN {X 0,Y 406.918,Z 853.268,A -85,B 0,C 180,E1 -11058.037,E2 -11058.037} C_VEL
LIN {X 0,Y 406.16,Z 861.76,A -85,B 0,C 180,E1 -11059.53,E2 -11059.53} C_VEL
LIN {X 0,Y 405.611,Z 868.502,A -85,B 0,C 180,E1 -11061.027,E2 -11061.027} C_VEL
LIN {X 0,Y 405.252,Z 873.879,A -85,B 0,C 180,E1 -11062.525,E2 -11062.525} C_VEL
LIN {X 0,Y 404.642,Z 878.142,A -85,B 0,C 180,E1 -11064.017,E2 -11064.017} C_VEL
LIN {X 0,Y 404.489,Z 880.367,A -85,B 0,C 180,E1 -11065.014,E2 -11065.014} C_VEL
LIN {X 0,Y 404.314,Z 882.187,A -85,B 0,C 180,E1 -11066.011,E2 -11066.011} C_VEL
LIN {X 0,Y 404.298,Z 883.542,A -85,B 0,C 180,E1 -11067.009,E2 -11067.009} C_VEL
LIN {X 0,Y 404.196,Z 885.112,A -85,B 0,C 180,E1 -11069.002,E2 -11069.002} C_VEL
LIN {X 0,Y 404.182,Z 885.341,A -85,B 0,C 180,E1 -11069.998,E2 -11069.998} C_VEL
LIN {X 0,Y 404.23,Z 884.593,A -85,B 0,C 180,E1 -11071.991,E2 -11071.991} C_VEL
LIN {X 0,Y 404.295,Z 883.654,A -85,B 0,C 180,E1 -11072.988,E2 -11072.988} C_VEL
LIN {X 0,Y 404.305,Z 882.348,A -85,B 0,C 180,E1 -11073.985,E2 -11073.985} C_VEL
LIN {X 0,Y 404.571,Z 879.545,A -85,B 0,C 180,E1 -11075.481,E2 -11075.481} C_VEL
LIN {X 0,Y 405.103,Z 875.715,A -85,B 0,C 180,E1 -11076.973,E2 -11076.973} C_VEL
LIN {X 0,Y 405.543,Z 870.324,A -85,B 0,C 180,E1 -11078.601,E2 -11078.601} C_VEL
LIN {X 0,Y 406.019,Z 863.445,A -85,B 0,C 180,E1 -11080.218,E2 -11080.218} C_VEL
LIN {X 0,Y 406.648,Z 856.898,A -85,B 0,C 180,E1 -11081.458,E2 -11081.458} C_VEL
LIN {X 0,Y 406.397,Z 853.21,A -85,B 0,C 180,E1 -11082.102,E2 -11082.102} C_VEL
LIN {X 0,Y 404.091,Z 847.085,A -85,B 0,C 180,E1 -11083.153,E2 -11083.153} C_VEL
LIN {X 0,Y 401.765,Z 840.426,A -85,B 0,C 180,E1 -11084.146,E2 -11084.146} C_VEL
LIN {X 0,Y 401.481,Z 835.856,A -85,B 0,C 180,E1 -11084.691,E2 -11084.691} C_VEL
LIN {X 0,Y 402.296,Z 825.054,A -85,B 0,C 180,E1 -11085.711,E2 -11085.711} C_VEL
LIN {X 0,Y 402.354,Z 820.138,A -85,B 0,C 180,E1 -11086.116,E2 -11086.116} C_VEL
LIN {X 0,Y 399.482,Z 810.237,A -85,B 0,C 180,E1 -11086.962,E2 -11086.962} C_VEL
LIN {X 0,Y 397.173,Z 803.014,A -85,B 0,C 180,E1 -11087.504,E2 -11087.504} C_VEL
LIN {X 0,Y 397.1,Z 803.017,A -85,B 0,C 180,E1 -11090.728,E2 -11090.728} C_VEL
LIN {X 0,Y 397.13,Z 803.019,A -85,B 0,C 180,E1 -11094.016,E2 -11094.016} C_VEL
LIN {X 0,Y 397.19,Z 803.009,A -85,B 0,C 180,E1 -11097.388,E2 -11097.388} C_VEL
LIN {X 0,Y 397.073,Z 803.022,A -85,B 0,C 180,E1 -11100.88,E2 -11100.88} C_VEL
LIN {X 0,Y 397.119,Z 803.019,A -85,B 0,C 180,E1 -11104.491,E2 -11104.491} C_VEL
LIN {X 0,Y 397.101,Z 803.024,A -85,B 0,C 180,E1 -11108.272,E2 -11108.272} C_VEL
LIN {X 0,Y 397.146,Z 803.015,A -85,B 0,C 180,E1 -11111.991,E2 -11111.991} C_VEL
LIN {X 0,Y 397.14,Z 803.013,A -85,B 0,C 180,E1 -11115.058,E2 -11115.058} C_VEL
LIN {X 0,Y 397.146,Z 803.01,A -85,B 0,C 180,E1 -11118.005,E2 -11118.005} C_VEL
LIN {X 0,Y 397.098,Z 803.013,A -85,B 0,C 180,E1 -11121.724,E2 -11121.724} C_VEL
LIN {X 0,Y 397.113,Z 803.011,A -85,B 0,C 180,E1 -11125.505,E2 -11125.505} C_VEL
LIN {X 0,Y 397.07,Z 803.019,A -85,B 0,C 180,E1 -11129.117,E2 -11129.117} C_VEL
LIN {X 0,Y 397.18,Z 803.012,A -85,B 0,C 180,E1 -11132.609,E2 -11132.609} C_VEL
LIN {X 0,Y 397.117,Z 803.014,A -85,B 0,C 180,E1 -11135.981,E2 -11135.981} C_VEL
LIN {X 0,Y 397.123,Z 803.012,A -85,B 0,C 180,E1 -11139.704,E2 -11139.704} C_VEL
LIN {X 0,Y 397.165,Z 803.014,A -85,B 0,C 180,E1 -11142.844,E2 -11142.844} C_VEL
LIN {X 0,Y 397.21,Z 803.004,A -85,B 0,C 180,E1 -11146.678,E2 -11146.678} C_VEL
LIN {X 0,Y 397.214,Z 803.001,A -85,B 0,C 180,E1 -11149.809,E2 -11149.809} C_VEL
LIN {X 0,Y 397.334,Z 802.991,A -85,B 0,C 180,E1 -11152.888,E2 -11152.888} C_VEL
LIN {X 0,Y 397.236,Z 803.005,A -85,B 0,C 180,E1 -11154.925,E2 -11154.925} C_VEL
LIN {X 0,Y 397.433,Z 802.979,A -85,B 0,C 180,E1 -11157.973,E2 -11157.973} C_VEL
LIN {X 0,Y 397.562,Z 802.964,A -85,B 0,C 180,E1 -11160,E2 -11160} C_VEL
LIN {X 0,Y 397.358,Z 802.989,A -85,B 0,C 180,E1 -11163.042,E2 -11163.042} C_VEL
LIN {X 0,Y 397.314,Z 802.992,A -85,B 0,C 180,E1 -11167.113,E2 -11167.113} C_VEL
LIN {X 0,Y 397.21,Z 803.005,A -85,B 0,C 180,E1 -11170.191,E2 -11170.191} C_VEL
LIN {X 0,Y 397.21,Z 803.001,A -85,B 0,C 180,E1 -11173.322,E2 -11173.322} C_VEL
LIN {X 0,Y 397.165,Z 803.011,A -85,B 0,C 180,E1 -11177.156,E2 -11177.156} C_VEL
LIN {X 0,Y 397.086,Z 803.021,A -85,B 0,C 180,E1 -11180.731,E2 -11180.731} C_VEL
LIN {X 0,Y 397.104,Z 803.023,A -85,B 0,C 180,E1 -11184.02,E2 -11184.02} C_VEL
LIN {X 0,Y 397.076,Z 803.021,A -85,B 0,C 180,E1 -11187.758,E2 -11187.758} C_VEL
LIN {X 0,Y 397.063,Z 803.024,A -85,B 0,C 180,E1 -11190.884,E2 -11190.884} C_VEL
LIN {X 0,Y 397.102,Z 803.021,A -85,B 0,C 180,E1 -11194.496,E2 -11194.496} C_VEL
LIN {X 0,Y 397.076,Z 803.025,A -85,B 0,C 180,E1 -11198.278,E2 -11198.278} C_VEL
LIN {X 0,Y 397.039,Z 803.024,A -85,B 0,C 180,E1 -11201.978,E2 -11201.978} C_VEL
LIN {X 0,Y 397.072,Z 803.022,A -85,B 0,C 180,E1 -11205.071,E2 -11205.071} C_VEL
LIN {X 0,Y 397.106,Z 803.168,A -85,B 0,C 180,E1 -11205.91,E2 -11205.91} C_VEL
LIN {X 0,Y 399.044,Z 812.603,A -85,B 0,C 180,E1 -11209.229,E2 -11209.229} C_VEL
LIN {X 0,Y 400.863,Z 822.453,A -85,B 0,C 180,E1 -11212.468,E2 -11212.468} C_VEL
LIN {X 0,Y 400.856,Z 826.698,A -85,B 0,C 180,E1 -11213.755,E2 -11213.755} C_VEL
LIN {X 0,Y 399.811,Z 839.802,A -85,B 0,C 180,E1 -11217.539,E2 -11217.539} C_VEL
LIN {X 0,Y 398.79,Z 854.23,A -85,B 0,C 180,E1 -11221.589,E2 -11221.589} C_VEL
LIN {X 0,Y 398.082,Z 866.343,A -85,B 0,C 180,E1 -11224.933,E2 -11224.933} C_VEL
LIN {X 0,Y 397.352,Z 880.178,A -85,B 0,C 180,E1 -11228.743,E2 -11228.743} C_VEL
LIN {X 0,Y 396.941,Z 890.889,A -85,B 0,C 180,E1 -11231.719,E2 -11231.719} C_VEL
LIN {X 0,Y 398.642,Z 906.61,A -85,B 0,C 180,E1 -11232.271,E2 -11232.271} C_VEL
LIN {X 0,Y 399.434,Z 919.112,A -85,B 0,C 180,E1 -11232.892,E2 -11232.892} C_VEL
LIN {X 0,Y 400.302,Z 929.423,A -85,B 0,C 180,E1 -11233.562,E2 -11233.562} C_VEL
LIN {X 0,Y 399.575,Z 940.857,A -85,B 0,C 180,E1 -11234.443,E2 -11234.443} C_VEL
LIN {X 0,Y 398.733,Z 951.361,A -85,B 0,C 180,E1 -11235.455,E2 -11235.455} C_VEL
LIN {X 0,Y 398.051,Z 960.468,A -85,B 0,C 180,E1 -11236.529,E2 -11236.529} C_VEL
LIN {X 0,Y 397.359,Z 969.052,A -85,B 0,C 180,E1 -11237.748,E2 -11237.748} C_VEL
LIN {X 0,Y 396.87,Z 976.53,A -85,B 0,C 180,E1 -11239.028,E2 -11239.028} C_VEL
LIN {X 0,Y 396.522,Z 983.93,A -85,B 0,C 180,E1 -11240.566,E2 -11240.566} C_VEL
LIN {X 0,Y 396.38,Z 988.945,A -85,B 0,C 180,E1 -11241.847,E2 -11241.847} C_VEL
LIN {X 0,Y 396.318,Z 993.446,A -85,B 0,C 180,E1 -11243.248,E2 -11243.248} C_VEL
LIN {X 0,Y 396.374,Z 997.598,A -85,B 0,C 180,E1 -11244.916,E2 -11244.916} C_VEL
LIN {X 0,Y 396.487,Z 999.55,A -85,B 0,C 180,E1 -11245.936,E2 -11245.936} C_VEL
LIN {X 0,Y 396.415,Z 1000.991,A -85,B 0,C 180,E1 -11246.953,E2 -11246.953} C_VEL
LIN {X 0,Y 396.428,Z 1002.027,A -85,B 0,C 180,E1 -11247.97,E2 -11247.97} C_VEL
LIN {X 0,Y 396.448,Z 1002.66,A -85,B 0,C 180,E1 -11248.986,E2 -11248.986} C_VEL
LIN {X 0,Y 396.466,Z 1002.886,A -85,B 0,C 180,E1 -11250.002,E2 -11250.002} C_VEL
LIN {X 0,Y 396.449,Z 1002.657,A -85,B 0,C 180,E1 -11251.018,E2 -11251.018} C_VEL
LIN {X 0,Y 396.429,Z 1002.021,A -85,B 0,C 180,E1 -11252.034,E2 -11252.034} C_VEL
LIN {X 0,Y 396.416,Z 1000.982,A -85,B 0,C 180,E1 -11253.051,E2 -11253.051} C_VEL
LIN {X 0,Y 396.488,Z 999.538,A -85,B 0,C 180,E1 -11254.068,E2 -11254.068} C_VEL
LIN {X 0,Y 396.302,Z 996.46,A -85,B 0,C 180,E1 -11255.599,E2 -11255.599} C_VEL
LIN {X 0,Y 396.311,Z 992.335,A -85,B 0,C 180,E1 -11257.133,E2 -11257.133} C_VEL
LIN {X 0,Y 396.441,Z 986.005,A -85,B 0,C 180,E1 -11258.925,E2 -11258.925} C_VEL
LIN {X 0,Y 396.748,Z 979.13,A -85,B 0,C 180,E1 -11260.463,E2 -11260.463} C_VEL
LIN {X 0,Y 397.313,Z 970.647,A -85,B 0,C 180,E1 -11261.998,E2 -11261.998} C_VEL
LIN {X 0,Y 398.111,Z 960.76,A -85,B 0,C 180,E1 -11263.429,E2 -11263.429} C_VEL
LIN {X 0,Y 398.785,Z 950.095,A -85,B 0,C 180,E1 -11264.677,E2 -11264.677} C_VEL
LIN {X 0,Y 399.676,Z 939.323,A -85,B 0,C 180,E1 -11265.687,E2 -11265.687} C_VEL
LIN {X 0,Y 400.266,Z 929.327,A -85,B 0,C 180,E1 -11266.443,E2 -11266.443} C_VEL
LIN {X 0,Y 399.328,Z 916.684,A -85,B 0,C 180,E1 -11267.238,E2 -11267.238} C_VEL
LIN {X 0,Y 398.329,Z 903.355,A -85,B 0,C 180,E1 -11267.855,E2 -11267.855} C_VEL
LIN {X 0,Y 396.949,Z 890.875,A -85,B 0,C 180,E1 -11268.284,E2 -11268.284} C_VEL
LIN {X 0,Y 397.346,Z 880.153,A -85,B 0,C 180,E1 -11271.261,E2 -11271.261} C_VEL
LIN {X 0,Y 398.01,Z 867.31,A -85,B 0,C 180,E1 -11274.797,E2 -11274.797} C_VEL
LIN {X 0,Y 398.651,Z 856.625,A -85,B 0,C 180,E1 -11277.741,E2 -11277.741} C_VEL
LIN {X 0,Y 399.548,Z 842.962,A -85,B 0,C 180,E1 -11281.555,E2 -11281.555} C_VEL
LIN {X 0,Y 400.448,Z 831.486,A -85,B 0,C 180,E1 -11284.831,E2 -11284.831} C_VEL
LIN {X 0,Y 400.955,Z 824.46,A -85,B 0,C 180,E1 -11286.896,E2 -11286.896} C_VEL
LIN {X 0,Y 400.092,Z 818.158,A -85,B 0,C 180,E1 -11288.903,E2 -11288.903} C_VEL
LIN {X 0,Y 398.203,Z 808.546,A -85,B 0,C 180,E1 -11292.16,E2 -11292.16} C_VEL
LIN {X 0,Y 397.089,Z 803.021,A -85,B 0,C 180,E1 -11294.174,E2 -11294.174} C_VEL
LIN {X 0,Y 397.032,Z 803.03,A -85,B 0,C 180,E1 -11298.028,E2 -11298.028} C_VEL
LIN {X 0,Y 397.091,Z 803.02,A -85,B 0,C 180,E1 -11301.147,E2 -11301.147} C_VEL
LIN {X 0,Y 397.093,Z 803.021,A -85,B 0,C 180,E1 -11304.504,E2 -11304.504} C_VEL
LIN {X 0,Y 397.077,Z 803.023,A -85,B 0,C 180,E1 -11307.928,E2 -11307.928} C_VEL
LIN {X 0,Y 397.118,Z 803.02,A -85,B 0,C 180,E1 -11310.295,E2 -11310.295} C_VEL
LIN {X 0,Y 397.07,Z 803.023,A -85,B 0,C 180,E1 -11313.737,E2 -11313.737} C_VEL
LIN {X 0,Y 397.105,Z 803.018,A -85,B 0,C 180,E1 -11317.085,E2 -11317.085} C_VEL
LIN {X 0,Y 397.085,Z 803.025,A -85,B 0,C 180,E1 -11320.35,E2 -11320.35} C_VEL
LIN {X 0,Y 397.08,Z 803.027,A -85,B 0,C 180,E1 -11322.13,E2 -11322.13} C_VEL
LIN {X 0,Y 400.858,Z 813.28,A -85,B 0,C 180,E1 -11323.061,E2 -11323.061} C_VEL
LIN {X 0,Y 403.12,Z 820.829,A -85,B 0,C 180,E1 -11323.803,E2 -11323.803} C_VEL
LIN {X 0,Y 402.589,Z 829.072,A -85,B 0,C 180,E1 -11324.51,E2 -11324.51} C_VEL
LIN {X 0,Y 402.022,Z 837.014,A -85,B 0,C 180,E1 -11325.316,E2 -11325.316} C_VEL
LIN {X 0,Y 401.39,Z 845.353,A -85,B 0,C 180,E1 -11326.327,E2 -11326.327} C_VEL
LIN {X 0,Y 400.623,Z 854.094,A -85,B 0,C 180,E1 -11327.59,E2 -11327.59} C_VEL
LIN {X 0,Y 399.899,Z 861.117,A -85,B 0,C 180,E1 -11328.853,E2 -11328.853} C_VEL
LIN {X 0,Y 399.446,Z 865.954,A -85,B 0,C 180,E1 -11329.866,E2 -11329.866} C_VEL
LIN {X 0,Y 399.054,Z 870.167,A -85,B 0,C 180,E1 -11330.88,E2 -11330.88} C_VEL
LIN {X 0,Y 398.256,Z 876.724,A -85,B 0,C 180,E1 -11332.904,E2 -11332.904} C_VEL
LIN {X 0,Y 397.817,Z 879.198,A -85,B 0,C 180,E1 -11333.915,E2 -11333.915} C_VEL
LIN {X 0,Y 397.746,Z 881.187,A -85,B 0,C 180,E1 -11334.931,E2 -11334.931} C_VEL
LIN {X 0,Y 397.415,Z 883.895,A -85,B 0,C 180,E1 -11336.959,E2 -11336.959} C_VEL
LIN {X 0,Y 397.102,Z 885.001,A -85,B 0,C 180,E1 -11338.986,E2 -11338.986} C_VEL
LIN {X 0,Y 397.056,Z 884.894,A -85,B 0,C 180,E1 -11340,E2 -11340} C_VEL
LIN {X 0,Y 397.059,Z 884.381,A -85,B 0,C 180,E1 -11341.014,E2 -11341.014} C_VEL
LIN {X 0,Y 396.95,Z 882.175,A -85,B 0,C 180,E1 -11343.045,E2 -11343.045} C_VEL
LIN {X 0,Y 397.167,Z 879.364,A -85,B 0,C 180,E1 -11344.567,E2 -11344.567} C_VEL
LIN {X 0,Y 397.438,Z 875.521,A -85,B 0,C 180,E1 -11346.091,E2 -11346.091} C_VEL
LIN {X 0,Y 397.738,Z 870.538,A -85,B 0,C 180,E1 -11347.616,E2 -11347.616} C_VEL
LIN {X 0,Y 398.097,Z 864.271,A -85,B 0,C 180,E1 -11349.142,E2 -11349.142} C_VEL
LIN {X 0,Y 398.619,Z 856.622,A -85,B 0,C 180,E1 -11350.668,E2 -11350.668} C_VEL
LIN {X 0,Y 399.135,Z 846.923,A -85,B 0,C 180,E1 -11352.198,E2 -11352.198} C_VEL
LIN {X 0,Y 399.837,Z 835.934,A -85,B 0,C 180,E1 -11353.597,E2 -11353.597} C_VEL
LIN {X 0,Y 400.388,Z 825.628,A -85,B 0,C 180,E1 -11354.657,E2 -11354.657} C_VEL
LIN {X 0,Y 400.755,Z 817.287,A -85,B 0,C 180,E1 -11355.368,E2 -11355.368} C_VEL
LIN {X 0,Y 397.9,Z 805.937,A -85,B 0,C 180,E1 -11356.284,E2 -11356.284} C_VEL
LIN {X 0,Y 397.17,Z 803.011,A -85,B 0,C 180,E1 -11356.509,E2 -11356.509} C_VEL
LIN {X 0,Y 397.103,Z 803.012,A -85,B 0,C 180,E1 -11360.278,E2 -11360.278} C_VEL
LIN {X 0,Y 397.109,Z 803.019,A -85,B 0,C 180,E1 -11364.02,E2 -11364.02} C_VEL
LIN {X 0,Y 397.067,Z 803.018,A -85,B 0,C 180,E1 -11367.4,E2 -11367.4} C_VEL
LIN {X 0,Y 397.104,Z 803.021,A -85,B 0,C 180,E1 -11369.862,E2 -11369.862} C_VEL
LIN {X 0,Y 397.122,Z 803.012,A -85,B 0,C 180,E1 -11373.717,E2 -11373.717} C_VEL
LIN {X 0,Y 397.093,Z 803.014,A -85,B 0,C 180,E1 -11377.207,E2 -11377.207} C_VEL
LIN {X 0,Y 397.061,Z 803.022,A -85,B 0,C 180,E1 -11380.437,E2 -11380.437} C_VEL
LIN {X 0,Y 397.104,Z 803.017,A -85,B 0,C 180,E1 -11383.648,E2 -11383.648} C_VEL
LIN {X 0,Y 397.107,Z 803.017,A -85,B 0,C 180,E1 -11386.521,E2 -11386.521} C_VEL
LIN {X 0,Y 397.093,Z 803.022,A -85,B 0,C 180,E1 -11390.419,E2 -11390.419} C_VEL
LIN {X 0,Y 397.103,Z 803.014,A -85,B 0,C 180,E1 -11393.004,E2 -11393.004} C_VEL
LIN {X 0,Y 397.125,Z 803.019,A -85,B 0,C 180,E1 -11396.281,E2 -11396.281} C_VEL
LIN {X 0,Y 397.112,Z 803.018,A -85,B 0,C 180,E1 -11400.134,E2 -11400.134} C_VEL
LIN {X 0,Y 397.2,Z 803.003,A -85,B 0,C 180,E1 -11402.609,E2 -11402.609} C_VEL
LIN {X 0,Y 397.135,Z 803.007,A -85,B 0,C 180,E1 -11405.98,E2 -11405.98} C_VEL
LIN {X 0,Y 397.145,Z 803.016,A -85,B 0,C 180,E1 -11409.703,E2 -11409.703} C_VEL
LIN {X 0,Y 397.18,Z 803.173,A -85,B 0,C 180,E1 -11412.616,E2 -11412.616} C_VEL
LIN {X 0,Y 400.956,Z 815.058,A -85,B 0,C 180,E1 -11413.532,E2 -11413.532} C_VEL
LIN {X 0,Y 402.48,Z 821.172,A -85,B 0,C 180,E1 -11414.07,E2 -11414.07} C_VEL
LIN {X 0,Y 401.718,Z 832.286,A -85,B 0,C 180,E1 -11415.044,E2 -11415.044} C_VEL
LIN {X 0,Y 400.98,Z 842.617,A -85,B 0,C 180,E1 -11416.182,E2 -11416.182} C_VEL
LIN {X 0,Y 400.334,Z 851.036,A -85,B 0,C 180,E1 -11417.322,E2 -11417.322} C_VEL
LIN {X 0,Y 399.61,Z 858.791,A -85,B 0,C 180,E1 -11418.587,E2 -11418.587} C_VEL
LIN {X 0,Y 398.959,Z 866.349,A -85,B 0,C 180,E1 -11420.109,E2 -11420.109} C_VEL
LIN {X 0,Y 398.49,Z 872.199,A -85,B 0,C 180,E1 -11421.58,E2 -11421.58} C_VEL
LIN {X 0,Y 398.126,Z 876.471,A -85,B 0,C 180,E1 -11422.9,E2 -11422.9} C_VEL
LIN {X 0,Y 397.587,Z 880.364,A -85,B 0,C 180,E1 -11424.419,E2 -11424.419} C_VEL
LIN {X 0,Y 397.307,Z 883.219,A -85,B 0,C 180,E1 -11425.941,E2 -11425.941} C_VEL
LIN {X 0,Y 397.283,Z 884.574,A -85,B 0,C 180,E1 -11426.956,E2 -11426.956} C_VEL
LIN {X 0,Y 397.178,Z 886.143,A -85,B 0,C 180,E1 -11428.984,E2 -11428.984} C_VEL
LIN {X 0,Y 397.16,Z 886.372,A -85,B 0,C 180,E1 -11429.998,E2 -11429.998} C_VEL
LIN {X 0,Y 397.224,Z 885.621,A -85,B 0,C 180,E1 -11432.026,E2 -11432.026} C_VEL
LIN {X 0,Y 397.298,Z 883.379,A -85,B 0,C 180,E1 -11434.056,E2 -11434.056} C_VEL
LIN {X 0,Y 397.578,Z 880.576,A -85,B 0,C 180,E1 -11435.577,E2 -11435.577} C_VEL
LIN {X 0,Y 398.136,Z 876.744,A -85,B 0,C 180,E1 -11437.096,E2 -11437.096} C_VEL
LIN {X 0,Y 398.62,Z 871.259,A -85,B 0,C 180,E1 -11438.776,E2 -11438.776} C_VEL
LIN {X 0,Y 399.133,Z 864.47,A -85,B 0,C 180,E1 -11440.396,E2 -11440.396} C_VEL
LIN {X 0,Y 399.902,Z 856.451,A -85,B 0,C 180,E1 -11441.915,E2 -11441.915} C_VEL
LIN {X 0,Y 400.574,Z 848.235,A -85,B 0,C 180,E1 -11443.182,E2 -11443.182} C_VEL
LIN {X 0,Y 401.287,Z 838.067,A -85,B 0,C 180,E1 -11444.45,E2 -11444.45} C_VEL
LIN {X 0,Y 401.481,Z 835.856,A -85,B 0,C 180,E1 -11444.691,E2 -11444.691} C_VEL
LIN {X 0,Y 401.189,Z 832.785,A -85,B 0,C 180,E1 -11445.042,E2 -11445.042} C_VEL
LIN {X 0,Y 399.065,Z 828.002,A -85,B 0,C 180,E1 -11445.629,E2 -11445.629} C_VEL
LIN {X 0,Y 395.868,Z 822.141,A -85,B 0,C 180,E1 -11446.306,E2 -11446.306} C_VEL
LIN {X 0,Y 395.11,Z 819.981,A -85,B 0,C 180,E1 -11446.516,E2 -11446.516} C_VEL
LIN {X 0,Y 392.004,Z 809.732,A -85,B 0,C 180,E1 -11447.395,E2 -11447.395} C_VEL
LIN {X 0,Y 390.127,Z 803.891,A -85,B 0,C 180,E1 -11447.831,E2 -11447.831} C_VEL
LIN {X 0,Y 390.053,Z 803.896,A -85,B 0,C 180,E1 -11451.12,E2 -11451.12} C_VEL
LIN {X 0,Y 390.076,Z 803.894,A -85,B 0,C 180,E1 -11454.479,E2 -11454.479} C_VEL
LIN {X 0,Y 390.112,Z 803.894,A -85,B 0,C 180,E1 -11457.928,E2 -11457.928} C_VEL
LIN {X 0,Y 390.018,Z 803.902,A -85,B 0,C 180,E1 -11461.502,E2 -11461.502} C_VEL
LIN {X 0,Y 390.061,Z 803.901,A -85,B 0,C 180,E1 -11464.023,E2 -11464.023} C_VEL
LIN {X 0,Y 390.039,Z 803.899,A -85,B 0,C 180,E1 -11467.549,E2 -11467.549} C_VEL
LIN {X 0,Y 390.074,Z 803.894,A -85,B 0,C 180,E1 -11470.824,E2 -11470.824} C_VEL
LIN {X 0,Y 390.116,Z 803.89,A -85,B 0,C 180,E1 -11473.895,E2 -11473.895} C_VEL
LIN {X 0,Y 390.107,Z 803.887,A -85,B 0,C 180,E1 -11476.796,E2 -11476.796} C_VEL
LIN {X 0,Y 390.067,Z 803.893,A -85,B 0,C 180,E1 -11479.562,E2 -11479.562} C_VEL
LIN {X 0,Y 390.048,Z 803.898,A -85,B 0,C 180,E1 -11482.444,E2 -11482.444} C_VEL
LIN {X 0,Y 390.054,Z 803.891,A -85,B 0,C 180,E1 -11486.044,E2 -11486.044} C_VEL
LIN {X 0,Y 390.038,Z 803.893,A -85,B 0,C 180,E1 -11489.866,E2 -11489.866} C_VEL
LIN {X 0,Y 390.099,Z 803.889,A -85,B 0,C 180,E1 -11493.231,E2 -11493.231} C_VEL
LIN {X 0,Y 390.091,Z 803.895,A -85,B 0,C 180,E1 -11496.749,E2 -11496.749} C_VEL
LIN {X 0,Y 390.088,Z 803.888,A -85,B 0,C 180,E1 -11499.982,E2 -11499.982} C_VEL
LIN {X 0,Y 390.121,Z 803.886,A -85,B 0,C 180,E1 -11503.247,E2 -11503.247} C_VEL
LIN {X 0,Y 390.178,Z 803.879,A -85,B 0,C 180,E1 -11506.561,E2 -11506.561} C_VEL
LIN {X 0,Y 390.163,Z 803.88,A -85,B 0,C 180,E1 -11509.623,E2 -11509.623} C_VEL
LIN {X 0,Y 390.285,Z 803.868,A -85,B 0,C 180,E1 -11512.758,E2 -11512.758} C_VEL
LIN {X 0,Y 390.208,Z 803.88,A -85,B 0,C 180,E1 -11514.833,E2 -11514.833} C_VEL
LIN {X 0,Y 390.402,Z 803.855,A -85,B 0,C 180,E1 -11517.937,E2 -11517.937} C_VEL
LIN {X 0,Y 390.532,Z 803.84,A -85,B 0,C 180,E1 -11520,E2 -11520} C_VEL
LIN {X 0,Y 390.293,Z 803.87,A -85,B 0,C 180,E1 -11523.097,E2 -11523.097} C_VEL
LIN {X 0,Y 390.284,Z 803.867,A -85,B 0,C 180,E1 -11526.203,E2 -11526.203} C_VEL
LIN {X 0,Y 390.191,Z 803.88,A -85,B 0,C 180,E1 -11529.329,E2 -11529.329} C_VEL
LIN {X 0,Y 390.161,Z 803.878,A -85,B 0,C 180,E1 -11532.483,E2 -11532.483} C_VEL
LIN {X 0,Y 390.122,Z 803.892,A -85,B 0,C 180,E1 -11535.678,E2 -11535.678} C_VEL
LIN {X 0,Y 390.087,Z 803.892,A -85,B 0,C 180,E1 -11538.923,E2 -11538.923} C_VEL
LIN {X 0,Y 390.021,Z 803.905,A -85,B 0,C 180,E1 -11542.235,E2 -11542.235} C_VEL
LIN {X 0,Y 390.034,Z 803.9,A -85,B 0,C 180,E1 -11545.723,E2 -11545.723} C_VEL
LIN {X 0,Y 390.017,Z 803.901,A -85,B 0,C 180,E1 -11549.113,E2 -11549.113} C_VEL
LIN {X 0,Y 390.027,Z 803.901,A -85,B 0,C 180,E1 -11552.723,E2 -11552.723} C_VEL
LIN {X 0,Y 390.028,Z 803.901,A -85,B 0,C 180,E1 -11555.824,E2 -11555.824} C_VEL
LIN {X 0,Y 390.022,Z 803.902,A -85,B 0,C 180,E1 -11559.214,E2 -11559.214} C_VEL
LIN {X 0,Y 390.017,Z 803.898,A -85,B 0,C 180,E1 -11562.374,E2 -11562.374} C_VEL
LIN {X 0,Y 390.059,Z 803.947,A -85,B 0,C 180,E1 -11565.477,E2 -11565.477} C_VEL
LIN {X 0,Y 391.937,Z 813.322,A -85,B 0,C 180,E1 -11568.862,E2 -11568.862} C_VEL
LIN {X 0,Y 393.607,Z 821.946,A -85,B 0,C 180,E1 -11571.78,E2 -11571.78} C_VEL
LIN {X 0,Y 394.018,Z 826.043,A -85,B 0,C 180,E1 -11573.088,E2 -11573.088} C_VEL
LIN {X 0,Y 393.11,Z 837.001,A -85,B 0,C 180,E1 -11576.346,E2 -11576.346} C_VEL
LIN {X 0,Y 392.261,Z 847.269,A -85,B 0,C 180,E1 -11579.317,E2 -11579.317} C_VEL
LIN {X 0,Y 391.496,Z 859.359,A -85,B 0,C 180,E1 -11582.759,E2 -11582.759} C_VEL
LIN {X 0,Y 390.758,Z 871.288,A -85,B 0,C 180,E1 -11586.126,E2 -11586.126} C_VEL
LIN {X 0,Y 390.08,Z 884.958,A -85,B 0,C 180,E1 -11589.984,E2 -11589.984} C_VEL
LIN {X 0,Y 389.873,Z 889.822,A -85,B 0,C 180,E1 -11591.376,E2 -11591.376} C_VEL
LIN {X 0,Y 391.664,Z 905.55,A -85,B 0,C 180,E1 -11591.945,E2 -11591.945} C_VEL
LIN {X 0,Y 392.459,Z 918.747,A -85,B 0,C 180,E1 -11592.619,E2 -11592.619} C_VEL
LIN {X 0,Y 393.337,Z 930.098,A -85,B 0,C 180,E1 -11593.391,E2 -11593.391} C_VEL
LIN {X 0,Y 392.549,Z 941.251,A -85,B 0,C 180,E1 -11594.291,E2 -11594.291} C_VEL
LIN {X 0,Y 391.711,Z 951.505,A -85,B 0,C 180,E1 -11595.322,E2 -11595.322} C_VEL
LIN {X 0,Y 390.989,Z 960.978,A -85,B 0,C 180,E1 -11596.489,E2 -11596.489} C_VEL
LIN {X 0,Y 390.274,Z 969.631,A -85,B 0,C 180,E1 -11597.786,E2 -11597.786} C_VEL
LIN {X 0,Y 389.69,Z 978.11,A -85,B 0,C 180,E1 -11599.349,E2 -11599.349} C_VEL
LIN {X 0,Y 389.393,Z 984.984,A -85,B 0,C 180,E1 -11600.916,E2 -11600.916} C_VEL
LIN {X 0,Y 389.241,Z 991.305,A -85,B 0,C 180,E1 -11602.741,E2 -11602.741} C_VEL
LIN {X 0,Y 389.246,Z 995.434,A -85,B 0,C 180,E1 -11604.303,E2 -11604.303} C_VEL
LIN {X 0,Y 389.432,Z 998.513,A -85,B 0,C 180,E1 -11605.862,E2 -11605.862} C_VEL
LIN {X 0,Y 389.379,Z 999.957,A -85,B 0,C 180,E1 -11606.898,E2 -11606.898} C_VEL
LIN {X 0,Y 389.393,Z 1000.994,A -85,B 0,C 180,E1 -11607.933,E2 -11607.933} C_VEL
LIN {X 0,Y 389.419,Z 1001.628,A -85,B 0,C 180,E1 -11608.968,E2 -11608.968} C_VEL
LIN {X 0,Y 389.441,Z 1001.854,A -85,B 0,C 180,E1 -11610.002,E2 -11610.002} C_VEL
LIN {X 0,Y 389.42,Z 1001.625,A -85,B 0,C 180,E1 -11611.036,E2 -11611.036} C_VEL
LIN {X 0,Y 389.394,Z 1000.987,A -85,B 0,C 180,E1 -11612.07,E2 -11612.07} C_VEL
LIN {X 0,Y 389.38,Z 999.947,A -85,B 0,C 180,E1 -11613.106,E2 -11613.106} C_VEL
LIN {X 0,Y 389.434,Z 998.499,A -85,B 0,C 180,E1 -11614.141,E2 -11614.141} C_VEL
LIN {X 0,Y 389.243,Z 995.418,A -85,B 0,C 180,E1 -11615.701,E2 -11615.701} C_VEL
LIN {X 0,Y 389.24,Z 991.287,A -85,B 0,C 180,E1 -11617.263,E2 -11617.263} C_VEL
LIN {X 0,Y 389.396,Z 984.957,A -85,B 0,C 180,E1 -11619.088,E2 -11619.088} C_VEL
LIN {X 0,Y 389.694,Z 978.075,A -85,B 0,C 180,E1 -11620.654,E2 -11620.654} C_VEL
LIN {X 0,Y 390.289,Z 969.59,A -85,B 0,C 180,E1 -11622.217,E2 -11622.217} C_VEL
LIN {X 0,Y 391.064,Z 960.932,A -85,B 0,C 180,E1 -11623.512,E2 -11623.512} C_VEL
LIN {X 0,Y 391.766,Z 950.234,A -85,B 0,C 180,E1 -11624.813,E2 -11624.813} C_VEL
LIN {X 0,Y 392.677,Z 939.716,A -85,B 0,C 180,E1 -11625.841,E2 -11625.841} C_VEL
LIN {X 0,Y 393.296,Z 929.979,A -85,B 0,C 180,E1 -11626.615,E2 -11626.615} C_VEL
LIN {X 0,Y 392.539,Z 918.699,A -85,B 0,C 180,E1 -11627.377,E2 -11627.377} C_VEL
LIN {X 0,Y 391.601,Z 905.45,A -85,B 0,C 180,E1 -11628.057,E2 -11628.057} C_VEL
LIN {X 0,Y 389.892,Z 889.696,A -85,B 0,C 180,E1 -11628.661,E2 -11628.661} C_VEL
LIN {X 0,Y 390.302,Z 879.129,A -85,B 0,C 180,E1 -11631.664,E2 -11631.664} C_VEL
LIN {X 0,Y 391.041,Z 866.329,A -85,B 0,C 180,E1 -11635.269,E2 -11635.269} C_VEL
LIN {X 0,Y 391.707,Z 855.031,A -85,B 0,C 180,E1 -11638.459,E2 -11638.459} C_VEL
LIN {X 0,Y 392.792,Z 841.029,A -85,B 0,C 180,E1 -11642.466,E2 -11642.466} C_VEL
LIN {X 0,Y 393.82,Z 828.732,A -85,B 0,C 180,E1 -11646.081,E2 -11646.081} C_VEL
LIN {X 0,Y 393.97,Z 824.616,A -85,B 0,C 180,E1 -11647.34,E2 -11647.34} C_VEL
LIN {X 0,Y 392.494,Z 816.18,A -85,B 0,C 180,E1 -11650.139,E2 -11650.139} C_VEL
LIN {X 0,Y 390.817,Z 807.763,A -85,B 0,C 180,E1 -11653.108,E2 -11653.108} C_VEL
LIN {X 0,Y 390.019,Z 803.906,A -85,B 0,C 180,E1 -11654.588,E2 -11654.588} C_VEL
LIN {X 0,Y 389.999,Z 803.906,A -85,B 0,C 180,E1 -11658.182,E2 -11658.182} C_VEL
LIN {X 0,Y 390.058,Z 803.897,A -85,B 0,C 180,E1 -11660.904,E2 -11660.904} C_VEL
LIN {X 0,Y 390.065,Z 803.896,A -85,B 0,C 180,E1 -11664.791,E2 -11664.791} C_VEL
LIN {X 0,Y 390.03,Z 803.901,A -85,B 0,C 180,E1 -11667.878,E2 -11667.878} C_VEL
LIN {X 0,Y 390.026,Z 803.902,A -85,B 0,C 180,E1 -11670.888,E2 -11670.888} C_VEL
LIN {X 0,Y 390.049,Z 803.901,A -85,B 0,C 180,E1 -11674.378,E2 -11674.378} C_VEL
LIN {X 0,Y 390.034,Z 803.9,A -85,B 0,C 180,E1 -11677.765,E2 -11677.765} C_VEL
LIN {X 0,Y 390.035,Z 803.903,A -85,B 0,C 180,E1 -11681.074,E2 -11681.074} C_VEL
LIN {X 0,Y 390.041,Z 803.901,A -85,B 0,C 180,E1 -11681.636,E2 -11681.636} C_VEL
LIN {X 0,Y 391.624,Z 808.241,A -85,B 0,C 180,E1 -11682.016,E2 -11682.016} C_VEL
LIN {X 0,Y 395.748,Z 819.736,A -85,B 0,C 180,E1 -11683.162,E2 -11683.162} C_VEL
LIN {X 0,Y 396.537,Z 823.237,A -85,B 0,C 180,E1 -11683.526,E2 -11683.526} C_VEL
LIN {X 0,Y 395.998,Z 830.997,A -85,B 0,C 180,E1 -11684.221,E2 -11684.221} C_VEL
LIN {X 0,Y 395.395,Z 839.004,A -85,B 0,C 180,E1 -11685.064,E2 -11685.064} C_VEL
LIN {X 0,Y 394.712,Z 847.199,A -85,B 0,C 180,E1 -11686.091,E2 -11686.091} C_VEL
LIN {X 0,Y 393.899,Z 855.828,A -85,B 0,C 180,E1 -11687.375,E2 -11687.375} C_VEL
LIN {X 0,Y 393.041,Z 864.009,A -85,B 0,C 180,E1 -11688.918,E2 -11688.918} C_VEL
LIN {X 0,Y 392.337,Z 870.306,A -85,B 0,C 180,E1 -11690.37,E2 -11690.37} C_VEL
LIN {X 0,Y 391.603,Z 876.672,A -85,B 0,C 180,E1 -11692.264,E2 -11692.264} C_VEL
LIN {X 0,Y 390.886,Z 880.537,A -85,B 0,C 180,E1 -11693.807,E2 -11693.807} C_VEL
LIN {X 0,Y 390.805,Z 882.508,A -85,B 0,C 180,E1 -11694.841,E2 -11694.841} C_VEL
LIN {X 0,Y 390.43,Z 885.11,A -85,B 0,C 180,E1 -11696.904,E2 -11696.904} C_VEL
LIN {X 0,Y 390.273,Z 885.826,A -85,B 0,C 180,E1 -11697.936,E2 -11697.936} C_VEL
LIN {X 0,Y 390.098,Z 886.15,A -85,B 0,C 180,E1 -11698.968,E2 -11698.968} C_VEL
LIN {X 0,Y 390.043,Z 885.997,A -85,B 0,C 180,E1 -11700,E2 -11700} C_VEL
LIN {X 0,Y 390.048,Z 885.447,A -85,B 0,C 180,E1 -11701.032,E2 -11701.032} C_VEL
LIN {X 0,Y 389.926,Z 883.137,A -85,B 0,C 180,E1 -11703.1,E2 -11703.1} C_VEL
LIN {X 0,Y 390.158,Z 880.253,A -85,B 0,C 180,E1 -11704.65,E2 -11704.65} C_VEL
LIN {X 0,Y 390.45,Z 876.332,A -85,B 0,C 180,E1 -11706.2,E2 -11706.2} C_VEL
LIN {X 0,Y 390.753,Z 871.27,A -85,B 0,C 180,E1 -11707.753,E2 -11707.753} C_VEL
LIN {X 0,Y 391.081,Z 866.116,A -85,B 0,C 180,E1 -11709.047,E2 -11709.047} C_VEL
LIN {X 0,Y 391.567,Z 858.568,A -85,B 0,C 180,E1 -11710.601,E2 -11710.601} C_VEL
LIN {X 0,Y 391.967,Z 850.78,A -85,B 0,C 180,E1 -11711.9,E2 -11711.9} C_VEL
LIN {X 0,Y 392.515,Z 842.492,A -85,B 0,C 180,E1 -11713.065,E2 -11713.065} C_VEL
LIN {X 0,Y 392.969,Z 834.934,A -85,B 0,C 180,E1 -11713.972,E2 -11713.972} C_VEL
LIN {X 0,Y 393.561,Z 824.322,A -85,B 0,C 180,E1 -11715.049,E2 -11715.049} C_VEL
LIN {X 0,Y 393.834,Z 818.697,A -85,B 0,C 180,E1 -11715.526,E2 -11715.526} C_VEL
LIN {X 0,Y 391.092,Z 807.643,A -85,B 0,C 180,E1 -11716.441,E2 -11716.441} C_VEL
LIN {X 0,Y 390.141,Z 803.887,A -85,B 0,C 180,E1 -11716.718,E2 -11716.718} C_VEL
LIN {X 0,Y 390.062,Z 803.889,A -85,B 0,C 180,E1 -11720.457,E2 -11720.457} C_VEL
LIN {X 0,Y 390.061,Z 803.894,A -85,B 0,C 180,E1 -11723.353,E2 -11723.353} C_VEL
LIN {X 0,Y 390.032,Z 803.891,A -85,B 0,C 180,E1 -11726.774,E2 -11726.774} C_VEL
LIN {X 0,Y 390.042,Z 803.896,A -85,B 0,C 180,E1 -11730.3,E2 -11730.3} C_VEL
LIN {X 0,Y 390.076,Z 803.894,A -85,B 0,C 180,E1 -11734.024,E2 -11734.024} C_VEL
LIN {X 0,Y 390.042,Z 803.895,A -85,B 0,C 180,E1 -11737.78,E2 -11737.78} C_VEL
LIN {X 0,Y 390.023,Z 803.897,A -85,B 0,C 180,E1 -11740.814,E2 -11740.814} C_VEL
LIN {X 0,Y 390.058,Z 803.898,A -85,B 0,C 180,E1 -11743.885,E2 -11743.885} C_VEL
LIN {X 0,Y 390.062,Z 803.893,A -85,B 0,C 180,E1 -11746.789,E2 -11746.789} C_VEL
LIN {X 0,Y 390.017,Z 803.9,A -85,B 0,C 180,E1 -11749.554,E2 -11749.554} C_VEL
LIN {X 0,Y 390.046,Z 803.897,A -85,B 0,C 180,E1 -11752.449,E2 -11752.449} C_VEL
LIN {X 0,Y 390.075,Z 803.896,A -85,B 0,C 180,E1 -11755.974,E2 -11755.974} C_VEL
LIN {X 0,Y 390.053,Z 803.894,A -85,B 0,C 180,E1 -11759.868,E2 -11759.868} C_VEL
LIN {X 0,Y 390.119,Z 803.883,A -85,B 0,C 180,E1 -11763.231,E2 -11763.231} C_VEL
LIN {X 0,Y 390.112,Z 803.89,A -85,B 0,C 180,E1 -11766.749,E2 -11766.749} C_VEL
LIN {X 0,Y 390.11,Z 803.894,A -85,B 0,C 180,E1 -11769.982,E2 -11769.982} C_VEL
LIN {X 0,Y 390.125,Z 803.896,A -85,B 0,C 180,E1 -11772.264,E2 -11772.264} C_VEL
LIN {X 0,Y 394.208,Z 816.812,A -85,B 0,C 180,E1 -11773.291,E2 -11773.291} C_VEL
LIN {X 0,Y 395.696,Z 822.409,A -85,B 0,C 180,E1 -11773.806,E2 -11773.806} C_VEL
LIN {X 0,Y 394.935,Z 833.322,A -85,B 0,C 180,E1 -11774.781,E2 -11774.781} C_VEL
LIN {X 0,Y 394.164,Z 843.652,A -85,B 0,C 180,E1 -11775.938,E2 -11775.938} C_VEL
LIN {X 0,Y 393.484,Z 852.07,A -85,B 0,C 180,E1 -11777.098,E2 -11777.098} C_VEL
LIN {X 0,Y 392.728,Z 859.825,A -85,B 0,C 180,E1 -11778.384,E2 -11778.384} C_VEL
LIN {X 0,Y 392.04,Z 867.383,A -85,B 0,C 180,E1 -11779.932,E2 -11779.932} C_VEL
LIN {X 0,Y 391.545,Z 873.212,A -85,B 0,C 180,E1 -11781.424,E2 -11781.424} C_VEL
LIN {X 0,Y 391.159,Z 877.503,A -85,B 0,C 180,E1 -11782.773,E2 -11782.773} C_VEL
LIN {X 0,Y 390.596,Z 881.396,A -85,B 0,C 180,E1 -11784.319,E2 -11784.319} C_VEL
LIN {X 0,Y 390.3,Z 884.251,A -85,B 0,C 180,E1 -11785.868,E2 -11785.868} C_VEL
LIN {X 0,Y 390.269,Z 885.606,A -85,B 0,C 180,E1 -11786.901,E2 -11786.901} C_VEL
LIN {X 0,Y 390.159,Z 887.173,A -85,B 0,C 180,E1 -11788.966,E2 -11788.966} C_VEL
LIN {X 0,Y 390.138,Z 887.403,A -85,B 0,C 180,E1 -11789.998,E2 -11789.998} C_VEL
LIN {X 0,Y 390.217,Z 886.65,A -85,B 0,C 180,E1 -11792.062,E2 -11792.062} C_VEL
LIN {X 0,Y 390.291,Z 884.409,A -85,B 0,C 180,E1 -11794.129,E2 -11794.129} C_VEL
LIN {X 0,Y 390.587,Z 881.606,A -85,B 0,C 180,E1 -11795.678,E2 -11795.678} C_VEL
LIN {X 0,Y 391.17,Z 877.773,A -85,B 0,C 180,E1 -11797.223,E2 -11797.223} C_VEL
LIN {X 0,Y 391.691,Z 872.234,A -85,B 0,C 180,E1 -11798.947,E2 -11798.947} C_VEL
LIN {X 0,Y 392.234,Z 865.498,A -85,B 0,C 180,E1 -11800.581,E2 -11800.581} C_VEL
LIN {X 0,Y 393.035,Z 857.479,A -85,B 0,C 180,E1 -11802.127,E2 -11802.127} C_VEL
LIN {X 0,Y 393.737,Z 849.263,A -85,B 0,C 180,E1 -11803.415,E2 -11803.415} C_VEL
LIN {X 0,Y 394.489,Z 839.094,A -85,B 0,C 180,E1 -11804.705,E2 -11804.705} C_VEL
LIN {X 0,Y 395.325,Z 828.967,A -85,B 0,C 180,E1 -11805.73,E2 -11805.73} C_VEL
LIN {X 0,Y 395.545,Z 821.6,A -85,B 0,C 180,E1 -11806.368,E2 -11806.368} C_VEL
LIN {X 0,Y 395.11,Z 819.981,A -85,B 0,C 180,E1 -11806.516,E2 -11806.516} C_VEL
LIN {X 0,Y 393.551,Z 817.004,A -85,B 0,C 180,E1 -11806.83,E2 -11806.83} C_VEL
LIN {X 0,Y 384.953,Z 809.038,A -85,B 0,C 180,E1 -11807.837,E2 -11807.837} C_VEL
LIN {X 0,Y 383.347,Z 805.87,A -85,B 0,C 180,E1 -11808.103,E2 -11808.103} C_VEL
LIN {X 0,Y 383.058,Z 804.771,A -85,B 0,C 180,E1 -11808.206,E2 -11808.206} C_VEL
LIN {X 0,Y 382.991,Z 804.778,A -85,B 0,C 180,E1 -11811.529,E2 -11811.529} C_VEL
LIN {X 0,Y 383.048,Z 804.769,A -85,B 0,C 180,E1 -11814.958,E2 -11814.958} C_VEL
LIN {X 0,Y 383.035,Z 804.772,A -85,B 0,C 180,E1 -11818.49,E2 -11818.49} C_VEL
LIN {X 0,Y 383.004,Z 804.78,A -85,B 0,C 180,E1 -11822.147,E2 -11822.147} C_VEL
LIN {X 0,Y 383.011,Z 804.775,A -85,B 0,C 180,E1 -11824.666,E2 -11824.666} C_VEL
LIN {X 0,Y 382.995,Z 804.78,A -85,B 0,C 180,E1 -11827.902,E2 -11827.902} C_VEL
LIN {X 0,Y 383.037,Z 804.769,A -85,B 0,C 180,E1 -11831.337,E2 -11831.337} C_VEL
LIN {X 0,Y 383.059,Z 804.772,A -85,B 0,C 180,E1 -11834.313,E2 -11834.313} C_VEL
LIN {X 0,Y 383.064,Z 804.762,A -85,B 0,C 180,E1 -11837.247,E2 -11837.247} C_VEL
LIN {X 0,Y 383.011,Z 804.776,A -85,B 0,C 180,E1 -11840.41,E2 -11840.41} C_VEL
LIN {X 0,Y 383.014,Z 804.773,A -85,B 0,C 180,E1 -11844.043,E2 -11844.043} C_VEL
LIN {X 0,Y 382.975,Z 804.777,A -85,B 0,C 180,E1 -11847.576,E2 -11847.576} C_VEL
LIN {X 0,Y 382.984,Z 804.774,A -85,B 0,C 180,E1 -11850.299,E2 -11850.299} C_VEL
LIN {X 0,Y 383.042,Z 804.774,A -85,B 0,C 180,E1 -11852.697,E2 -11852.697} C_VEL
LIN {X 0,Y 383.037,Z 804.771,A -85,B 0,C 180,E1 -11855.039,E2 -11855.039} C_VEL
LIN {X 0,Y 382.977,Z 804.777,A -85,B 0,C 180,E1 -11858.468,E2 -11858.468} C_VEL
LIN {X 0,Y 383.047,Z 804.768,A -85,B 0,C 180,E1 -11861.826,E2 -11861.826} C_VEL
LIN {X 0,Y 383.095,Z 804.76,A -85,B 0,C 180,E1 -11865.118,E2 -11865.118} C_VEL
LIN {X 0,Y 383.093,Z 804.763,A -85,B 0,C 180,E1 -11868.358,E2 -11868.358} C_VEL
LIN {X 0,Y 383.246,Z 804.744,A -85,B 0,C 180,E1 -11871.975,E2 -11871.975} C_VEL
LIN {X 0,Y 383.18,Z 804.755,A -85,B 0,C 180,E1 -11874.738,E2 -11874.738} C_VEL
LIN {X 0,Y 383.37,Z 804.731,A -85,B 0,C 180,E1 -11877.899,E2 -11877.899} C_VEL
LIN {X 0,Y 383.501,Z 804.716,A -85,B 0,C 180,E1 -11880,E2 -11880} C_VEL
LIN {X 0,Y 383.23,Z 804.751,A -85,B 0,C 180,E1 -11883.154,E2 -11883.154} C_VEL
LIN {X 0,Y 383.242,Z 804.744,A -85,B 0,C 180,E1 -11886.317,E2 -11886.317} C_VEL
LIN {X 0,Y 383.205,Z 804.748,A -85,B 0,C 180,E1 -11888.437,E2 -11888.437} C_VEL
LIN {X 0,Y 383.09,Z 804.764,A -85,B 0,C 180,E1 -11891.642,E2 -11891.642} C_VEL
LIN {X 0,Y 383.094,Z 804.763,A -85,B 0,C 180,E1 -11894.882,E2 -11894.882} C_VEL
LIN {X 0,Y 383.072,Z 804.771,A -85,B 0,C 180,E1 -11898.173,E2 -11898.173} C_VEL
LIN {X 0,Y 382.975,Z 804.78,A -85,B 0,C 180,E1 -11901.532,E2 -11901.532} C_VEL
LIN {X 0,Y 382.975,Z 804.777,A -85,B 0,C 180,E1 -11904.966,E2 -11904.966} C_VEL
LIN {X 0,Y 382.97,Z 804.782,A -85,B 0,C 180,E1 -11908.498,E2 -11908.498} C_VEL
LIN {X 0,Y 382.994,Z 804.779,A -85,B 0,C 180,E1 -11912.151,E2 -11912.151} C_VEL
LIN {X 0,Y 382.997,Z 804.777,A -85,B 0,C 180,E1 -11914.67,E2 -11914.67} C_VEL
LIN {X 0,Y 382.978,Z 804.781,A -85,B 0,C 180,E1 -11917.904,E2 -11917.904} C_VEL
LIN {X 0,Y 382.947,Z 804.782,A -85,B 0,C 180,E1 -11921.352,E2 -11921.352} C_VEL
LIN {X 0,Y 382.976,Z 804.776,A -85,B 0,C 180,E1 -11924.304,E2 -11924.304} C_VEL
LIN {X 0,Y 382.986,Z 804.785,A -85,B 0,C 180,E1 -11925.046,E2 -11925.046} C_VEL
LIN {X 0,Y 384.898,Z 814,A -85,B 0,C 180,E1 -11928.472,E2 -11928.472} C_VEL
LIN {X 0,Y 386.724,Z 823.757,A -85,B 0,C 180,E1 -11931.841,E2 -11931.841} C_VEL
LIN {X 0,Y 387.041,Z 827.941,A -85,B 0,C 180,E1 -11933.189,E2 -11933.189} C_VEL
LIN {X 0,Y 385.957,Z 840.179,A -85,B 0,C 180,E1 -11936.891,E2 -11936.891} C_VEL
LIN {X 0,Y 384.952,Z 852.351,A -85,B 0,C 180,E1 -11940.469,E2 -11940.469} C_VEL
LIN {X 0,Y 384.138,Z 864.384,A -85,B 0,C 180,E1 -11943.957,E2 -11943.957} C_VEL
LIN {X 0,Y 383.4,Z 876.201,A -85,B 0,C 180,E1 -11947.362,E2 -11947.362} C_VEL
LIN {X 0,Y 382.849,Z 887.7,A -85,B 0,C 180,E1 -11950.708,E2 -11950.708} C_VEL
LIN {X 0,Y 382.823,Z 888.755,A -85,B 0,C 180,E1 -11951.02,E2 -11951.02} C_VEL
LIN {X 0,Y 384.653,Z 904.57,A -85,B 0,C 180,E1 -11951.608,E2 -11951.608} C_VEL
LIN {X 0,Y 385.496,Z 916.769,A -85,B 0,C 180,E1 -11952.24,E2 -11952.24} C_VEL
LIN {X 0,Y 386.097,Z 927.436,A -85,B 0,C 180,E1 -11952.952,E2 -11952.952} C_VEL
LIN {X 0,Y 386.267,Z 932.554,A -85,B 0,C 180,E1 -11953.35,E2 -11953.35} C_VEL
LIN {X 0,Y 385.287,Z 944.281,A -85,B 0,C 180,E1 -11954.394,E2 -11954.394} C_VEL
LIN {X 0,Y 384.336,Z 955.497,A -85,B 0,C 180,E1 -11955.652,E2 -11955.652} C_VEL
LIN {X 0,Y 383.782,Z 963.592,A -85,B 0,C 180,E1 -11956.769,E2 -11956.769} C_VEL
LIN {X 0,Y 383.059,Z 971.63,A -85,B 0,C 180,E1 -11958.09,E2 -11958.09} C_VEL
LIN {X 0,Y 382.548,Z 979.532,A -85,B 0,C 180,E1 -11959.683,E2 -11959.683} C_VEL
LIN {X 0,Y 382.252,Z 986.852,A -85,B 0,C 180,E1 -11961.544,E2 -11961.544} C_VEL
LIN {X 0,Y 382.175,Z 992.021,A -85,B 0,C 180,E1 -11963.234,E2 -11963.234} C_VEL
LIN {X 0,Y 382.238,Z 995.516,A -85,B 0,C 180,E1 -11964.727,E2 -11964.727} C_VEL
LIN {X 0,Y 382.379,Z 997.475,A -85,B 0,C 180,E1 -11965.786,E2 -11965.786} C_VEL
LIN {X 0,Y 382.341,Z 998.923,A -85,B 0,C 180,E1 -11966.841,E2 -11966.841} C_VEL
LIN {X 0,Y 382.358,Z 999.961,A -85,B 0,C 180,E1 -11967.895,E2 -11967.895} C_VEL
LIN {X 0,Y 382.39,Z 1000.596,A -85,B 0,C 180,E1 -11968.949,E2 -11968.949} C_VEL
LIN {X 0,Y 382.416,Z 1000.823,A -85,B 0,C 180,E1 -11970.002,E2 -11970.002} C_VEL
LIN {X 0,Y 382.39,Z 1000.592,A -85,B 0,C 180,E1 -11971.055,E2 -11971.055} C_VEL
LIN {X 0,Y 382.359,Z 999.953,A -85,B 0,C 180,E1 -11972.109,E2 -11972.109} C_VEL
LIN {X 0,Y 382.342,Z 998.912,A -85,B 0,C 180,E1 -11973.163,E2 -11973.163} C_VEL
LIN {X 0,Y 382.381,Z 997.46,A -85,B 0,C 180,E1 -11974.218,E2 -11974.218} C_VEL
LIN {X 0,Y 382.185,Z 994.376,A -85,B 0,C 180,E1 -11975.807,E2 -11975.807} C_VEL
LIN {X 0,Y 382.188,Z 990.242,A -85,B 0,C 180,E1 -11977.398,E2 -11977.398} C_VEL
LIN {X 0,Y 382.354,Z 983.908,A -85,B 0,C 180,E1 -11979.257,E2 -11979.257} C_VEL
LIN {X 0,Y 382.665,Z 977.023,A -85,B 0,C 180,E1 -11980.852,E2 -11980.852} C_VEL
LIN {X 0,Y 383.252,Z 968.531,A -85,B 0,C 180,E1 -11982.445,E2 -11982.445} C_VEL
LIN {X 0,Y 384.033,Z 959.867,A -85,B 0,C 180,E1 -11983.765,E2 -11983.765} C_VEL
LIN {X 0,Y 384.828,Z 949.177,A -85,B 0,C 180,E1 -11985.086,E2 -11985.086} C_VEL
LIN {X 0,Y 385.948,Z 937.219,A -85,B 0,C 180,E1 -11986.26,E2 -11986.26} C_VEL
LIN {X 0,Y 386.331,Z 930.711,A -85,B 0,C 180,E1 -11986.787,E2 -11986.787} C_VEL
LIN {X 0,Y 385.665,Z 920.262,A -85,B 0,C 180,E1 -11987.54,E2 -11987.54} C_VEL
LIN {X 0,Y 384.852,Z 907.086,A -85,B 0,C 180,E1 -11988.267,E2 -11988.267} C_VEL
LIN {X 0,Y 383.208,Z 891.059,A -85,B 0,C 180,E1 -11989.025,E2 -11989.025} C_VEL
LIN {X 0,Y 382.844,Z 888.043,A -85,B 0,C 180,E1 -11989.192,E2 -11989.192} C_VEL
LIN {X 0,Y 383.408,Z 876.173,A -85,B 0,C 180,E1 -11992.641,E2 -11992.641} C_VEL
LIN {X 0,Y 384.121,Z 864.338,A -85,B 0,C 180,E1 -11996.049,E2 -11996.049} C_VEL
LIN {X 0,Y 384.85,Z 853.854,A -85,B 0,C 180,E1 -11999.081,E2 -11999.081} C_VEL
LIN {X 0,Y 385.85,Z 841.174,A -85,B 0,C 180,E1 -12002.803,E2 -12002.803} C_VEL
LIN {X 0,Y 386.965,Z 828.879,A -85,B 0,C 180,E1 -12006.5,E2 -12006.5} C_VEL
LIN {X 0,Y 386.856,Z 824.721,A -85,B 0,C 180,E1 -12007.828,E2 -12007.828} C_VEL
LIN {X 0,Y 385.092,Z 815.247,A -85,B 0,C 180,E1 -12011.074,E2 -12011.074} C_VEL
LIN {X 0,Y 383.106,Z 805.417,A -85,B 0,C 180,E1 -12014.695,E2 -12014.695} C_VEL
LIN {X 0,Y 382.969,Z 804.784,A -85,B 0,C 180,E1 -12015.048,E2 -12015.048} C_VEL
LIN {X 0,Y 382.959,Z 804.783,A -85,B 0,C 180,E1 -12018.803,E2 -12018.803} C_VEL
LIN {X 0,Y 382.994,Z 804.78,A -85,B 0,C 180,E1 -12022.099,E2 -12022.099} C_VEL
LIN {X 0,Y 383.02,Z 804.773,A -85,B 0,C 180,E1 -12025.662,E2 -12025.662} C_VEL
LIN {X 0,Y 382.983,Z 804.779,A -85,B 0,C 180,E1 -12029.081,E2 -12029.081} C_VEL
LIN {X 0,Y 382.969,Z 804.782,A -85,B 0,C 180,E1 -12032.691,E2 -12032.691} C_VEL
LIN {X 0,Y 383.007,Z 804.777,A -85,B 0,C 180,E1 -12036.191,E2 -12036.191} C_VEL
LIN {X 0,Y 383.03,Z 804.776,A -85,B 0,C 180,E1 -12039.597,E2 -12039.597} C_VEL
LIN {X 0,Y 382.992,Z 804.785,A -85,B 0,C 180,E1 -12041.095,E2 -12041.095} C_VEL
